LIN {X 0,Y 246.856,Z 370.948,A -85,B 0,C 180,E1 -19029.765,E2 -19029.765} C_VEL
LIN {X 0,Y 247.348,Z 370.564,A -85,B 0,C 180,E1 -19032.995,E2 -19032.995} C_VEL
LIN {X 0,Y 247.895,Z 369.406,A -85,B 0,C 180,E1 -19035.136,E2 -19035.136} C_VEL
LIN {X 0,Y 249.122,Z 366.297,A -85,B 0,C 180,E1 -19038.384,E2 -19038.384} C_VEL
LIN {X 0,Y 250.289,Z 363.157,A -85,B 0,C 180,E1 -19040.597,E2 -19040.597} C_VEL
LIN {X 0,Y 252.077,Z 357.887,A -85,B 0,C 180,E1 -19043.344,E2 -19043.344} C_VEL
LIN {X 0,Y 254.344,Z 351.173,A -85,B 0,C 180,E1 -19045.993,E2 -19045.993} C_VEL
LIN {X 0,Y 256.495,Z 344.263,A -85,B 0,C 180,E1 -19048.149,E2 -19048.149} C_VEL
LIN {X 0,Y 259.318,Z 334.726,A -85,B 0,C 180,E1 -19050.481,E2 -19050.481} C_VEL
LIN {X 0,Y 261.847,Z 325.143,A -85,B 0,C 180,E1 -19052.343,E2 -19052.343} C_VEL
LIN {X 0,Y 264.393,Z 314.469,A -85,B 0,C 180,E1 -19053.979,E2 -19053.979} C_VEL
LIN {X 0,Y 266.72,Z 302.445,A -85,B 0,C 180,E1 -19055.418,E2 -19055.418} C_VEL
LIN {X 0,Y 268.611,Z 289.891,A -85,B 0,C 180,E1 -19056.566,E2 -19056.566} C_VEL
LIN {X 0,Y 269.924,Z 277.78,A -85,B 0,C 180,E1 -19057.366,E2 -19057.366} C_VEL
LIN {X 0,Y 270.894,Z 265.944,A -85,B 0,C 180,E1 -19057.879,E2 -19057.879} C_VEL
LIN {X 0,Y 273.87,Z 206.722,A -85,B 0,C 180,E1 -19059.638,E2 -19059.638} C_VEL
LIN {X 0,Y 268.916,Z 195.841,A -85,B 0,C 180,E1 -19060.94,E2 -19060.94} C_VEL
LIN {X 0,Y 263.621,Z 185.772,A -85,B 0,C 180,E1 -19062.367,E2 -19062.367} C_VEL
LIN {X 0,Y 258.048,Z 176.312,A -85,B 0,C 180,E1 -19063.953,E2 -19063.953} C_VEL
LIN {X 0,Y 254.517,Z 171.077,A -85,B 0,C 180,E1 -19064.995,E2 -19064.995} C_VEL
LIN {X 0,Y 252.04,Z 167.296,A -85,B 0,C 180,E1 -19065.776,E2 -19065.776} C_VEL
LIN {X 0,Y 250.053,Z 164.997,A -85,B 0,C 180,E1 -19066.386,E2 -19066.386} C_VEL
LIN {X 0,Y 249.299,Z 163,A -85,B 0,C 180,E1 -19066.708,E2 -19066.708} C_VEL
LIN {X 0,Y 249.238,Z 162.44,A -85,B 0,C 180,E1 -19067.171,E2 -19067.171} C_VEL
LIN {X 0,Y 249.422,Z 162.416,A -85,B 0,C 180,E1 -19071.902,E2 -19071.902} C_VEL
LIN {X 0,Y 249.267,Z 162.431,A -85,B 0,C 180,E1 -19075.149,E2 -19075.149} C_VEL
LIN {X 0,Y 249.636,Z 162.383,A -85,B 0,C 180,E1 -19078.272,E2 -19078.272} C_VEL
LIN {X 0,Y 249.448,Z 162.41,A -85,B 0,C 180,E1 -19079.172,E2 -19079.172} C_VEL
LIN {X 0,Y 248.655,Z 162.514,A -85,B 0,C 180,E1 -19080.058,E2 -19080.058} C_VEL
LIN {X 0,Y 246.082,Z 162.842,A -85,B 0,C 180,E1 -19081.801,E2 -19081.801} C_VEL
LIN {X 0,Y 243.415,Z 163.173,A -85,B 0,C 180,E1 -19083.583,E2 -19083.583} C_VEL
LIN {X 0,Y 242.311,Z 163.302,A -85,B 0,C 180,E1 -19084.974,E2 -19084.974} C_VEL
LIN {X 0,Y 242.252,Z 163.303,A -85,B 0,C 180,E1 -19085.447,E2 -19085.447} C_VEL
LIN {X 0,Y 242.373,Z 163.288,A -85,B 0,C 180,E1 -19088.337,E2 -19088.337} C_VEL
LIN {X 0,Y 242.112,Z 163.324,A -85,B 0,C 180,E1 -19093.429,E2 -19093.429} C_VEL
LIN {X 0,Y 242.097,Z 163.326,A -85,B 0,C 180,E1 -19096.877,E2 -19096.877} C_VEL
LIN {X 0,Y 241.976,Z 163.342,A -85,B 0,C 180,E1 -19102.184,E2 -19102.184} C_VEL
LIN {X 0,Y 241.991,Z 163.342,A -85,B 0,C 180,E1 -19105.827,E2 -19105.827} C_VEL
LIN {X 0,Y 241.968,Z 163.346,A -85,B 0,C 180,E1 -19109.59,E2 -19109.59} C_VEL
LIN {X 0,Y 241.984,Z 163.343,A -85,B 0,C 180,E1 -19113.493,E2 -19113.493} C_VEL
LIN {X 0,Y 241.992,Z 163.337,A -85,B 0,C 180,E1 -19117.582,E2 -19117.582} C_VEL
LIN {X 0,Y 241.913,Z 163.348,A -85,B 0,C 180,E1 -19121.929,E2 -19121.929} C_VEL
LIN {X 0,Y 241.966,Z 163.485,A -85,B 0,C 180,E1 -19122.861,E2 -19122.861} C_VEL
LIN {X 0,Y 243.695,Z 168.875,A -85,B 0,C 180,E1 -19126.198,E2 -19126.198} C_VEL
LIN {X 0,Y 246.03,Z 176.729,A -85,B 0,C 180,E1 -19130.47,E2 -19130.47} C_VEL
LIN {X 0,Y 248.775,Z 181.528,A -85,B 0,C 180,E1 -19131.44,E2 -19131.44} C_VEL
LIN {X 0,Y 250.887,Z 185.194,A -85,B 0,C 180,E1 -19132.142,E2 -19132.142} C_VEL
LIN {X 0,Y 253.14,Z 189.148,A -85,B 0,C 180,E1 -19132.863,E2 -19132.863} C_VEL
LIN {X 0,Y 258.623,Z 199.785,A -85,B 0,C 180,E1 -19134.545,E2 -19134.545} C_VEL
LIN {X 0,Y 262.961,Z 209.455,A -85,B 0,C 180,E1 -19135.836,E2 -19135.836} C_VEL
LIN {X 0,Y 264.023,Z 212.177,A -85,B 0,C 180,E1 -19136.15,E2 -19136.15} C_VEL
LIN {X 0,Y 266.656,Z 231.739,A -85,B 0,C 180,E1 -19137.415,E2 -19137.415} C_VEL
LIN {X 0,Y 267.038,Z 237.313,A -85,B 0,C 180,E1 -19137.701,E2 -19137.701} C_VEL
LIN {X 0,Y 264.288,Z 288.303,A -85,B 0,C 180,E1 -19139.27,E2 -19139.27} C_VEL
LIN {X 0,Y 262.866,Z 301.195,A -85,B 0,C 180,E1 -19139.913,E2 -19139.913} C_VEL
LIN {X 0,Y 260.719,Z 314.41,A -85,B 0,C 180,E1 -19140.862,E2 -19140.862} C_VEL
LIN {X 0,Y 258.383,Z 326.026,A -85,B 0,C 180,E1 -19142.017,E2 -19142.017} C_VEL
LIN {X 0,Y 256.04,Z 336.044,A -85,B 0,C 180,E1 -19143.289,E2 -19143.289} C_VEL
LIN {X 0,Y 253.243,Z 346.542,A -85,B 0,C 180,E1 -19144.961,E2 -19144.961} C_VEL
LIN {X 0,Y 250.418,Z 356.075,A -85,B 0,C 180,E1 -19146.863,E2 -19146.863} C_VEL
LIN {X 0,Y 247.988,Z 364.065,A -85,B 0,C 180,E1 -19148.86,E2 -19148.86} C_VEL
LIN {X 0,Y 245.836,Z 371.131,A -85,B 0,C 180,E1 -19151.044,E2 -19151.044} C_VEL
LIN {X 0,Y 243.985,Z 376.967,A -85,B 0,C 180,E1 -19153.258,E2 -19153.258} C_VEL
LIN {X 0,Y 242.22,Z 382.172,A -85,B 0,C 180,E1 -19155.721,E2 -19155.721} C_VEL
LIN {X 0,Y 241.046,Z 386.261,A -85,B 0,C 180,E1 -19158.223,E2 -19158.223} C_VEL
LIN {X 0,Y 240.142,Z 390.101,A -85,B 0,C 180,E1 -19161.585,E2 -19161.585} C_VEL
LIN {X 0,Y 239.898,Z 391.414,A -85,B 0,C 180,E1 -19163.269,E2 -19163.269} C_VEL
LIN {X 0,Y 239.808,Z 392.369,A -85,B 0,C 180,E1 -19165.167,E2 -19165.167} C_VEL
LIN {X 0,Y 239.971,Z 392.844,A -85,B 0,C 180,E1 -19168.321,E2 -19168.321} C_VEL
LIN {X 0,Y 240.02,Z 392.522,A -85,B 0,C 180,E1 -19169.999,E2 -19169.999} C_VEL
LIN {X 0,Y 239.988,Z 391.764,A -85,B 0,C 180,E1 -19171.677,E2 -19171.677} C_VEL
LIN {X 0,Y 239.94,Z 390.556,A -85,B 0,C 180,E1 -19173.357,E2 -19173.357} C_VEL
LIN {X 0,Y 239.915,Z 388.833,A -85,B 0,C 180,E1 -19175.126,E2 -19175.126} C_VEL
LIN {X 0,Y 240.072,Z 385.603,A -85,B 0,C 180,E1 -19177.569,E2 -19177.569} C_VEL
LIN {X 0,Y 240.467,Z 381.156,A -85,B 0,C 180,E1 -19180.099,E2 -19180.099} C_VEL
LIN {X 0,Y 241.155,Z 375.461,A -85,B 0,C 180,E1 -19182.624,E2 -19182.624} C_VEL
LIN {X 0,Y 242.422,Z 368.321,A -85,B 0,C 180,E1 -19185.124,E2 -19185.124} C_VEL
LIN {X 0,Y 243.817,Z 359.891,A -85,B 0,C 180,E1 -19187.472,E2 -19187.472} C_VEL
LIN {X 0,Y 245.472,Z 350.125,A -85,B 0,C 180,E1 -19189.657,E2 -19189.657} C_VEL
LIN {X 0,Y 247.269,Z 339.949,A -85,B 0,C 180,E1 -19191.464,E2 -19191.464} C_VEL
LIN {X 0,Y 249.026,Z 328.652,A -85,B 0,C 180,E1 -19193.052,E2 -19193.052} C_VEL
LIN {X 0,Y 250.727,Z 316.016,A -85,B 0,C 180,E1 -19194.421,E2 -19194.421} C_VEL
LIN {X 0,Y 252.123,Z 303.843,A -85,B 0,C 180,E1 -19195.377,E2 -19195.377} C_VEL
LIN {X 0,Y 253.166,Z 290.677,A -85,B 0,C 180,E1 -19196.092,E2 -19196.092} C_VEL
LIN {X 0,Y 254.777,Z 250.055,A -85,B 0,C 180,E1 -19197.365,E2 -19197.365} C_VEL
LIN {X 0,Y 255.305,Z 232.614,A -85,B 0,C 180,E1 -19197.902,E2 -19197.902} C_VEL
LIN {X 0,Y 250.199,Z 193.129,A -85,B 0,C 180,E1 -19199.733,E2 -19199.733} C_VEL
LIN {X 0,Y 245.773,Z 180.605,A -85,B 0,C 180,E1 -19200.64,E2 -19200.64} C_VEL
LIN {X 0,Y 243.127,Z 168.039,A -85,B 0,C 180,E1 -19205.318,E2 -19205.318} C_VEL
LIN {X 0,Y 242.041,Z 163.337,A -85,B 0,C 180,E1 -19207.221,E2 -19207.221} C_VEL
LIN {X 0,Y 241.938,Z 163.352,A -85,B 0,C 180,E1 -19211.921,E2 -19211.921} C_VEL
LIN {X 0,Y 241.934,Z 163.348,A -85,B 0,C 180,E1 -19216.57,E2 -19216.57} C_VEL
LIN {X 0,Y 241.956,Z 163.345,A -85,B 0,C 180,E1 -19220.28,E2 -19220.28} C_VEL
LIN {X 0,Y 242.004,Z 163.339,A -85,B 0,C 180,E1 -19224.491,E2 -19224.491} C_VEL
LIN {X 0,Y 241.975,Z 163.343,A -85,B 0,C 180,E1 -19228.479,E2 -19228.479} C_VEL
LIN {X 0,Y 242.009,Z 163.337,A -85,B 0,C 180,E1 -19232.312,E2 -19232.312} C_VEL
LIN {X 0,Y 242.056,Z 163.327,A -85,B 0,C 180,E1 -19236.015,E2 -19236.015} C_VEL
LIN {X 0,Y 242.025,Z 163.338,A -85,B 0,C 180,E1 -19239.606,E2 -19239.606} C_VEL
LIN {X 0,Y 242.114,Z 163.321,A -85,B 0,C 180,E1 -19243.315,E2 -19243.315} C_VEL
LIN {X 0,Y 242.182,Z 163.316,A -85,B 0,C 180,E1 -19248.279,E2 -19248.279} C_VEL
LIN {X 0,Y 242.424,Z 163.278,A -85,B 0,C 180,E1 -19251.665,E2 -19251.665} C_VEL
LIN {X 0,Y 242.258,Z 163.307,A -85,B 0,C 180,E1 -19255.006,E2 -19255.006} C_VEL
LIN {X 0,Y 242.635,Z 163.26,A -85,B 0,C 180,E1 -19258.339,E2 -19258.339} C_VEL
LIN {X 0,Y 242.634,Z 163.251,A -85,B 0,C 180,E1 -19261.659,E2 -19261.659} C_VEL
LIN {X 0,Y 242.426,Z 163.287,A -85,B 0,C 180,E1 -19266.703,E2 -19266.703} C_VEL
LIN {X 0,Y 242.311,Z 163.299,A -85,B 0,C 180,E1 -19270.021,E2 -19270.021} C_VEL
LIN {X 0,Y 242.163,Z 163.312,A -85,B 0,C 180,E1 -19275.14,E2 -19275.14} C_VEL
LIN {X 0,Y 242.07,Z 163.332,A -85,B 0,C 180,E1 -19278.623,E2 -19278.623} C_VEL
LIN {X 0,Y 242.038,Z 163.334,A -85,B 0,C 180,E1 -19282.176,E2 -19282.176} C_VEL
LIN {X 0,Y 242.062,Z 163.318,A -85,B 0,C 180,E1 -19285.838,E2 -19285.838} C_VEL
LIN {X 0,Y 242.026,Z 163.332,A -85,B 0,C 180,E1 -19289.58,E2 -19289.58} C_VEL
LIN {X 0,Y 241.987,Z 163.336,A -85,B 0,C 180,E1 -19293.49,E2 -19293.49} C_VEL
LIN {X 0,Y 242.015,Z 163.328,A -85,B 0,C 180,E1 -19297.576,E2 -19297.576} C_VEL
LIN {X 0,Y 242.038,Z 163.335,A -85,B 0,C 180,E1 -19301.9,E2 -19301.9} C_VEL
LIN {X 0,Y 242.02,Z 163.33,A -85,B 0,C 180,E1 -19306.548,E2 -19306.548} C_VEL
LIN {X 0,Y 242.024,Z 163.336,A -85,B 0,C 180,E1 -19310.295,E2 -19310.295} C_VEL
LIN {X 0,Y 242.032,Z 163.328,A -85,B 0,C 180,E1 -19314.498,E2 -19314.498} C_VEL
LIN {X 0,Y 241.971,Z 163.342,A -85,B 0,C 180,E1 -19318.48,E2 -19318.48} C_VEL
LIN {X 0,Y 242.004,Z 163.338,A -85,B 0,C 180,E1 -19322.313,E2 -19322.313} C_VEL
LIN {X 0,Y 242.053,Z 163.333,A -85,B 0,C 180,E1 -19326.016,E2 -19326.016} C_VEL
LIN {X 0,Y 242.033,Z 163.337,A -85,B 0,C 180,E1 -19329.609,E2 -19329.609} C_VEL
LIN {X 0,Y 242.159,Z 163.323,A -85,B 0,C 180,E1 -19333.279,E2 -19333.279} C_VEL
LIN {X 0,Y 242.183,Z 163.318,A -85,B 0,C 180,E1 -19338.281,E2 -19338.281} C_VEL
LIN {X 0,Y 242.431,Z 163.288,A -85,B 0,C 180,E1 -19341.667,E2 -19341.667} C_VEL
LIN {X 0,Y 242.259,Z 163.311,A -85,B 0,C 180,E1 -19345.008,E2 -19345.008} C_VEL
LIN {X 0,Y 242.634,Z 163.261,A -85,B 0,C 180,E1 -19348.341,E2 -19348.341} C_VEL
LIN {X 0,Y 242.634,Z 163.261,A -85,B 0,C 180,E1 -19351.661,E2 -19351.661} C_VEL
LIN {X 0,Y 242.416,Z 163.29,A -85,B 0,C 180,E1 -19357.183,E2 -19357.183} C_VEL
LIN {X 0,Y 243.5,Z 166.231,A -85,B 0,C 180,E1 -19357.438,E2 -19357.438} C_VEL
LIN {X 0,Y 250.973,Z 183.621,A -85,B 0,C 180,E1 -19358.835,E2 -19358.835} C_VEL
LIN {X 0,Y 256.265,Z 198.404,A -85,B 0,C 180,E1 -19359.848,E2 -19359.848} C_VEL
LIN {X 0,Y 253.616,Z 268.159,A -85,B 0,C 180,E1 -19361.996,E2 -19361.996} C_VEL
LIN {X 0,Y 252.675,Z 281.492,A -85,B 0,C 180,E1 -19362.723,E2 -19362.723} C_VEL
LIN {X 0,Y 251.611,Z 294.331,A -85,B 0,C 180,E1 -19363.766,E2 -19363.766} C_VEL
LIN {X 0,Y 250.2,Z 306.198,A -85,B 0,C 180,E1 -19365.061,E2 -19365.061} C_VEL
LIN {X 0,Y 248.544,Z 317.502,A -85,B 0,C 180,E1 -19366.638,E2 -19366.638} C_VEL
LIN {X 0,Y 246.824,Z 327.773,A -85,B 0,C 180,E1 -19368.442,E2 -19368.442} C_VEL
LIN {X 0,Y 245.209,Z 337.341,A -85,B 0,C 180,E1 -19370.556,E2 -19370.556} C_VEL
LIN {X 0,Y 243.795,Z 345.266,A -85,B 0,C 180,E1 -19372.711,E2 -19372.711} C_VEL
LIN {X 0,Y 242.442,Z 352.962,A -85,B 0,C 180,E1 -19375.315,E2 -19375.315} C_VEL
LIN {X 0,Y 241.421,Z 358.656,A -85,B 0,C 180,E1 -19377.761,E2 -19377.761} C_VEL
LIN {X 0,Y 240.608,Z 363.958,A -85,B 0,C 180,E1 -19380.742,E2 -19380.742} C_VEL
LIN {X 0,Y 239.939,Z 367.864,A -85,B 0,C 180,E1 -19383.817,E2 -19383.817} C_VEL
LIN {X 0,Y 239.728,Z 369.62,A -85,B 0,C 180,E1 -19385.898,E2 -19385.898} C_VEL
LIN {X 0,Y 239.652,Z 370.797,A -85,B 0,C 180,E1 -19388.014,E2 -19388.014} C_VEL
LIN {X 0,Y 239.809,Z 371.334,A -85,B 0,C 180,E1 -19390.363,E2 -19390.363} C_VEL
LIN {X 0,Y 240.26,Z 370.996,A -85,B 0,C 180,E1 -19393.007,E2 -19393.007} C_VEL
LIN {X 0,Y 240.933,Z 369.713,A -85,B 0,C 180,E1 -19395.568,E2 -19395.568} C_VEL
LIN {X 0,Y 242.293,Z 366.515,A -85,B 0,C 180,E1 -19398.954,E2 -19398.954} C_VEL
LIN {X 0,Y 244.033,Z 361.975,A -85,B 0,C 180,E1 -19402.042,E2 -19402.042} C_VEL
LIN {X 0,Y 246.091,Z 356.398,A -85,B 0,C 180,E1 -19404.785,E2 -19404.785} C_VEL
LIN {X 0,Y 248.697,Z 349.008,A -85,B 0,C 180,E1 -19407.527,E2 -19407.527} C_VEL
LIN {X 0,Y 251.218,Z 341.32,A -85,B 0,C 180,E1 -19409.765,E2 -19409.765} C_VEL
LIN {X 0,Y 253.797,Z 332.678,A -85,B 0,C 180,E1 -19411.78,E2 -19411.78} C_VEL
LIN {X 0,Y 256.518,Z 322.579,A -85,B 0,C 180,E1 -19413.646,E2 -19413.646} C_VEL
LIN {X 0,Y 259.316,Z 310.658,A -85,B 0,C 180,E1 -19415.375,E2 -19415.375} C_VEL
LIN {X 0,Y 261.448,Z 299.381,A -85,B 0,C 180,E1 -19416.642,E2 -19416.642} C_VEL
LIN {X 0,Y 263.307,Z 286.431,A -85,B 0,C 180,E1 -19417.749,E2 -19417.749} C_VEL
LIN {X 0,Y 264.683,Z 273.244,A -85,B 0,C 180,E1 -19418.529,E2 -19418.529} C_VEL
LIN {X 0,Y 265.814,Z 256.165,A -85,B 0,C 180,E1 -19419.114,E2 -19419.114} C_VEL
LIN {X 0,Y 268.28,Z 208.894,A -85,B 0,C 180,E1 -19420.539,E2 -19420.539} C_VEL
LIN {X 0,Y 263.182,Z 197.855,A -85,B 0,C 180,E1 -19421.947,E2 -19421.947} C_VEL
LIN {X 0,Y 256.603,Z 185.498,A -85,B 0,C 180,E1 -19423.86,E2 -19423.86} C_VEL
LIN {X 0,Y 250.777,Z 176.379,A -85,B 0,C 180,E1 -19425.651,E2 -19425.651} C_VEL
LIN {X 0,Y 248.175,Z 172.649,A -85,B 0,C 180,E1 -19426.49,E2 -19426.49} C_VEL
LIN {X 0,Y 245.905,Z 169.455,A -85,B 0,C 180,E1 -19427.246,E2 -19427.246} C_VEL
LIN {X 0,Y 245.166,Z 168.24,A -85,B 0,C 180,E1 -19427.513,E2 -19427.513} C_VEL
LIN {X 0,Y 243.09,Z 165.951,A -85,B 0,C 180,E1 -19428.22,E2 -19428.22} C_VEL
LIN {X 0,Y 242.265,Z 163.59,A -85,B 0,C 180,E1 -19428.603,E2 -19428.603} C_VEL
LIN {X 0,Y 242.221,Z 163.314,A -85,B 0,C 180,E1 -19429.13,E2 -19429.13} C_VEL
LIN {X 0,Y 242.376,Z 163.295,A -85,B 0,C 180,E1 -19431.665,E2 -19431.665} C_VEL
LIN {X 0,Y 242.401,Z 163.291,A -85,B 0,C 180,E1 -19433.341,E2 -19433.341} C_VEL
LIN {X 0,Y 242.622,Z 163.257,A -85,B 0,C 180,E1 -19438.341,E2 -19438.341} C_VEL
LIN {X 0,Y 242.619,Z 163.26,A -85,B 0,C 180,E1 -19441.661,E2 -19441.661} C_VEL
LIN {X 0,Y 242.252,Z 163.303,A -85,B 0,C 180,E1 -19445.447,E2 -19445.447} C_VEL
LIN {X 0,Y 241.65,Z 163.373,A -85,B 0,C 180,E1 -19446.836,E2 -19446.836} C_VEL
LIN {X 0,Y 240.066,Z 163.577,A -85,B 0,C 180,E1 -19448.199,E2 -19448.199} C_VEL
LIN {X 0,Y 236.239,Z 164.051,A -85,B 0,C 180,E1 -19450.942,E2 -19450.942} C_VEL
LIN {X 0,Y 235.141,Z 164.187,A -85,B 0,C 180,E1 -19452.376,E2 -19452.376} C_VEL
LIN {X 0,Y 235.045,Z 164.194,A -85,B 0,C 180,E1 -19452.862,E2 -19452.862} C_VEL
LIN {X 0,Y 235.055,Z 164.203,A -85,B 0,C 180,E1 -19456.903,E2 -19456.903} C_VEL
LIN {X 0,Y 234.961,Z 164.217,A -85,B 0,C 180,E1 -19461.987,E2 -19461.987} C_VEL
LIN {X 0,Y 234.927,Z 164.215,A -85,B 0,C 180,E1 -19466.664,E2 -19466.664} C_VEL
LIN {X 0,Y 234.9,Z 164.218,A -85,B 0,C 180,E1 -19470.573,E2 -19470.573} C_VEL
LIN {X 0,Y 234.934,Z 164.212,A -85,B 0,C 180,E1 -19474.638,E2 -19474.638} C_VEL
LIN {X 0,Y 234.917,Z 164.217,A -85,B 0,C 180,E1 -19478.935,E2 -19478.935} C_VEL
LIN {X 0,Y 234.904,Z 164.425,A -85,B 0,C 180,E1 -19480.88,E2 -19480.88} C_VEL
LIN {X 0,Y 237.096,Z 171.042,A -85,B 0,C 180,E1 -19485.351,E2 -19485.351} C_VEL
LIN {X 0,Y 238.745,Z 176.397,A -85,B 0,C 180,E1 -19488.409,E2 -19488.409} C_VEL
LIN {X 0,Y 241.757,Z 181.355,A -85,B 0,C 180,E1 -19489.56,E2 -19489.56} C_VEL
LIN {X 0,Y 243.391,Z 184.153,A -85,B 0,C 180,E1 -19490.167,E2 -19490.167} C_VEL
LIN {X 0,Y 246.439,Z 189.214,A -85,B 0,C 180,E1 -19491.224,E2 -19491.224} C_VEL
LIN {X 0,Y 250.836,Z 197.293,A -85,B 0,C 180,E1 -19492.705,E2 -19492.705} C_VEL
LIN {X 0,Y 256.982,Z 210.263,A -85,B 0,C 180,E1 -19494.654,E2 -19494.654} C_VEL
LIN {X 0,Y 259.057,Z 215.917,A -85,B 0,C 180,E1 -19495.329,E2 -19495.329} C_VEL
LIN {X 0,Y 261.248,Z 233.871,A -85,B 0,C 180,E1 -19496.508,E2 -19496.508} C_VEL
LIN {X 0,Y 261.539,Z 238.959,A -85,B 0,C 180,E1 -19496.77,E2 -19496.77} C_VEL
LIN {X 0,Y 258.697,Z 288.182,A -85,B 0,C 180,E1 -19498.306,E2 -19498.306} C_VEL
LIN {X 0,Y 257.222,Z 300.955,A -85,B 0,C 180,E1 -19498.954,E2 -19498.954} C_VEL
LIN {X 0,Y 255.004,Z 314.123,A -85,B 0,C 180,E1 -19499.916,E2 -19499.916} C_VEL
LIN {X 0,Y 252.191,Z 327.24,A -85,B 0,C 180,E1 -19501.266,E2 -19501.266} C_VEL
LIN {X 0,Y 249.779,Z 336.941,A -85,B 0,C 180,E1 -19502.564,E2 -19502.564} C_VEL
LIN {X 0,Y 246.856,Z 347.196,A -85,B 0,C 180,E1 -19504.267,E2 -19504.267} C_VEL
LIN {X 0,Y 243.914,Z 356.501,A -85,B 0,C 180,E1 -19506.209,E2 -19506.209} C_VEL
LIN {X 0,Y 240.995,Z 365.586,A -85,B 0,C 180,E1 -19508.62,E2 -19508.62} C_VEL
LIN {X 0,Y 238.534,Z 372.957,A -85,B 0,C 180,E1 -19511.088,E2 -19511.088} C_VEL
LIN {X 0,Y 236.524,Z 378.907,A -85,B 0,C 180,E1 -19513.603,E2 -19513.603} C_VEL
LIN {X 0,Y 234.799,Z 383.635,A -85,B 0,C 180,E1 -19516.145,E2 -19516.145} C_VEL
LIN {X 0,Y 233.762,Z 387.273,A -85,B 0,C 180,E1 -19518.73,E2 -19518.73} C_VEL
LIN {X 0,Y 233.09,Z 389.922,A -85,B 0,C 180,E1 -19521.328,E2 -19521.328} C_VEL
LIN {X 0,Y 232.819,Z 391.19,A -85,B 0,C 180,E1 -19523.064,E2 -19523.064} C_VEL
LIN {X 0,Y 232.719,Z 392.172,A -85,B 0,C 180,E1 -19525.272,E2 -19525.272} C_VEL
LIN {X 0,Y 232.897,Z 392.499,A -85,B 0,C 180,E1 -19528.27,E2 -19528.27} C_VEL
LIN {X 0,Y 232.948,Z 392.138,A -85,B 0,C 180,E1 -19529.999,E2 -19529.999} C_VEL
LIN {X 0,Y 232.917,Z 391.316,A -85,B 0,C 180,E1 -19531.728,E2 -19531.728} C_VEL
LIN {X 0,Y 232.858,Z 390.072,A -85,B 0,C 180,E1 -19533.46,E2 -19533.46} C_VEL
LIN {X 0,Y 232.841,Z 387.374,A -85,B 0,C 180,E1 -19536.063,E2 -19536.063} C_VEL
LIN {X 0,Y 233.143,Z 383.613,A -85,B 0,C 180,E1 -19538.668,E2 -19538.668} C_VEL
LIN {X 0,Y 233.641,Z 378.67,A -85,B 0,C 180,E1 -19541.274,E2 -19541.274} C_VEL
LIN {X 0,Y 234.605,Z 372.417,A -85,B 0,C 180,E1 -19543.865,E2 -19543.865} C_VEL
LIN {X 0,Y 235.978,Z 364.596,A -85,B 0,C 180,E1 -19546.434,E2 -19546.434} C_VEL
LIN {X 0,Y 237.534,Z 355.633,A -85,B 0,C 180,E1 -19548.772,E2 -19548.772} C_VEL
LIN {X 0,Y 239.34,Z 345.658,A -85,B 0,C 180,E1 -19550.856,E2 -19550.856} C_VEL
LIN {X 0,Y 241.052,Z 335.864,A -85,B 0,C 180,E1 -19552.498,E2 -19552.498} C_VEL
LIN {X 0,Y 242.723,Z 325.281,A -85,B 0,C 180,E1 -19553.913,E2 -19553.913} C_VEL
LIN {X 0,Y 244.427,Z 312.638,A -85,B 0,C 180,E1 -19555.207,E2 -19555.207} C_VEL
LIN {X 0,Y 245.806,Z 299.367,A -85,B 0,C 180,E1 -19556.191,E2 -19556.191} C_VEL
LIN {X 0,Y 246.761,Z 285.995,A -85,B 0,C 180,E1 -19556.823,E2 -19556.823} C_VEL
LIN {X 0,Y 248.696,Z 233.355,A -85,B 0,C 180,E1 -19558.477,E2 -19558.477} C_VEL
LIN {X 0,Y 243.803,Z 195.193,A -85,B 0,C 180,E1 -19560.307,E2 -19560.307} C_VEL
LIN {X 0,Y 238.46,Z 180.289,A -85,B 0,C 180,E1 -19561.437,E2 -19561.437} C_VEL
LIN {X 0,Y 236.274,Z 169.835,A -85,B 0,C 180,E1 -19565.451,E2 -19565.451} C_VEL
LIN {X 0,Y 234.974,Z 164.217,A -85,B 0,C 180,E1 -19567.707,E2 -19567.707} C_VEL
LIN {X 0,Y 234.884,Z 164.231,A -85,B 0,C 180,E1 -19571.579,E2 -19571.579} C_VEL
LIN {X 0,Y 234.895,Z 164.226,A -85,B 0,C 180,E1 -19575.894,E2 -19575.894} C_VEL
LIN {X 0,Y 234.883,Z 164.225,A -85,B 0,C 180,E1 -19578.831,E2 -19578.831} C_VEL
LIN {X 0,Y 234.918,Z 164.222,A -85,B 0,C 180,E1 -19581.077,E2 -19581.077} C_VEL
LIN {X 0,Y 234.941,Z 164.22,A -85,B 0,C 180,E1 -19585.363,E2 -19585.363} C_VEL
LIN {X 0,Y 234.931,Z 164.22,A -85,B 0,C 180,E1 -19589.431,E2 -19589.431} C_VEL
LIN {X 0,Y 234.993,Z 164.212,A -85,B 0,C 180,E1 -19593.792,E2 -19593.792} C_VEL
LIN {X 0,Y 235.005,Z 164.211,A -85,B 0,C 180,E1 -19598.968,E2 -19598.968} C_VEL
LIN {X 0,Y 235.077,Z 164.196,A -85,B 0,C 180,E1 -19604.39,E2 -19604.39} C_VEL
LIN {X 0,Y 235.236,Z 164.179,A -85,B 0,C 180,E1 -19609.672,E2 -19609.672} C_VEL
LIN {X 0,Y 235.401,Z 164.156,A -85,B 0,C 180,E1 -19613.14,E2 -19613.14} C_VEL
LIN {X 0,Y 235.594,Z 164.137,A -85,B 0,C 180,E1 -19618.29,E2 -19618.29} C_VEL
LIN {X 0,Y 235.594,Z 164.127,A -85,B 0,C 180,E1 -19621.708,E2 -19621.708} C_VEL
LIN {X 0,Y 235.4,Z 164.164,A -85,B 0,C 180,E1 -19626.858,E2 -19626.858} C_VEL
LIN {X 0,Y 235.235,Z 164.182,A -85,B 0,C 180,E1 -19630.326,E2 -19630.326} C_VEL
LIN {X 0,Y 235.11,Z 164.19,A -85,B 0,C 180,E1 -19635.606,E2 -19635.606} C_VEL
LIN {X 0,Y 235.005,Z 164.209,A -85,B 0,C 180,E1 -19639.205,E2 -19639.205} C_VEL
LIN {X 0,Y 234.973,Z 164.209,A -85,B 0,C 180,E1 -19642.881,E2 -19642.881} C_VEL
LIN {X 0,Y 234.966,Z 164.207,A -85,B 0,C 180,E1 -19646.657,E2 -19646.657} C_VEL
LIN {X 0,Y 234.928,Z 164.219,A -85,B 0,C 180,E1 -19650.567,E2 -19650.567} C_VEL
LIN {X 0,Y 234.956,Z 164.208,A -85,B 0,C 180,E1 -19654.632,E2 -19654.632} C_VEL
LIN {X 0,Y 234.992,Z 164.207,A -85,B 0,C 180,E1 -19658.961,E2 -19658.961} C_VEL
LIN {X 0,Y 234.992,Z 164.21,A -85,B 0,C 180,E1 -19663.46,E2 -19663.46} C_VEL
LIN {X 0,Y 234.998,Z 164.21,A -85,B 0,C 180,E1 -19668.387,E2 -19668.387} C_VEL
LIN {X 0,Y 234.981,Z 164.213,A -85,B 0,C 180,E1 -19671.092,E2 -19671.092} C_VEL
LIN {X 0,Y 234.956,Z 164.211,A -85,B 0,C 180,E1 -19675.367,E2 -19675.367} C_VEL
LIN {X 0,Y 234.964,Z 164.215,A -85,B 0,C 180,E1 -19680.158,E2 -19680.158} C_VEL
LIN {X 0,Y 234.989,Z 164.214,A -85,B 0,C 180,E1 -19683.794,E2 -19683.794} C_VEL
LIN {X 0,Y 235.007,Z 164.212,A -85,B 0,C 180,E1 -19688.97,E2 -19688.97} C_VEL
LIN {X 0,Y 235.092,Z 164.202,A -85,B 0,C 180,E1 -19693.06,E2 -19693.06} C_VEL
LIN {X 0,Y 235.143,Z 164.196,A -85,B 0,C 180,E1 -19697.925,E2 -19697.925} C_VEL
LIN {X 0,Y 235.387,Z 164.167,A -85,B 0,C 180,E1 -19701.415,E2 -19701.415} C_VEL
LIN {X 0,Y 235.402,Z 164.167,A -85,B 0,C 180,E1 -19703.142,E2 -19703.142} C_VEL
LIN {X 0,Y 235.593,Z 164.138,A -85,B 0,C 180,E1 -19708.292,E2 -19708.292} C_VEL
LIN {X 0,Y 235.593,Z 164.138,A -85,B 0,C 180,E1 -19711.71,E2 -19711.71} C_VEL
LIN {X 0,Y 235.359,Z 164.169,A -85,B 0,C 180,E1 -19716.43,E2 -19716.43} C_VEL
LIN {X 0,Y 236.439,Z 167.089,A -85,B 0,C 180,E1 -19716.675,E2 -19716.675} C_VEL
LIN {X 0,Y 243.5,Z 182.958,A -85,B 0,C 180,E1 -19718.04,E2 -19718.04} C_VEL
LIN {X 0,Y 249.65,Z 199.841,A -85,B 0,C 180,E1 -19719.265,E2 -19719.265} C_VEL
LIN {X 0,Y 246.975,Z 268.023,A -85,B 0,C 180,E1 -19721.415,E2 -19721.415} C_VEL
LIN {X 0,Y 245.998,Z 281.897,A -85,B 0,C 180,E1 -19722.19,E2 -19722.19} C_VEL
LIN {X 0,Y 244.851,Z 294.888,A -85,B 0,C 180,E1 -19723.276,E2 -19723.276} C_VEL
LIN {X 0,Y 243.365,Z 306.967,A -85,B 0,C 180,E1 -19724.638,E2 -19724.638} C_VEL
LIN {X 0,Y 241.617,Z 318.399,A -85,B 0,C 180,E1 -19726.288,E2 -19726.288} C_VEL
LIN {X 0,Y 239.875,Z 328.509,A -85,B 0,C 180,E1 -19728.138,E2 -19728.138} C_VEL
LIN {X 0,Y 238.107,Z 338.524,A -85,B 0,C 180,E1 -19730.44,E2 -19730.44} C_VEL
LIN {X 0,Y 236.55,Z 347.149,A -85,B 0,C 180,E1 -19732.927,E2 -19732.927} C_VEL
LIN {X 0,Y 235.238,Z 354.064,A -85,B 0,C 180,E1 -19735.437,E2 -19735.437} C_VEL
LIN {X 0,Y 234.329,Z 359.113,A -85,B 0,C 180,E1 -19737.703,E2 -19737.703} C_VEL
LIN {X 0,Y 233.491,Z 364.396,A -85,B 0,C 180,E1 -19740.778,E2 -19740.778} C_VEL
LIN {X 0,Y 232.829,Z 368.27,A -85,B 0,C 180,E1 -19743.948,E2 -19743.948} C_VEL
LIN {X 0,Y 232.556,Z 370.658,A -85,B 0,C 180,E1 -19747.188,E2 -19747.188} C_VEL
LIN {X 0,Y 232.635,Z 371.499,A -85,B 0,C 180,E1 -19749.378,E2 -19749.378} C_VEL
LIN {X 0,Y 232.864,Z 371.647,A -85,B 0,C 180,E1 -19751.605,E2 -19751.605} C_VEL
LIN {X 0,Y 233.374,Z 371.16,A -85,B 0,C 180,E1 -19753.841,E2 -19753.841} C_VEL
LIN {X 0,Y 234.076,Z 369.838,A -85,B 0,C 180,E1 -19756.327,E2 -19756.327} C_VEL
LIN {X 0,Y 235.596,Z 366.555,A -85,B 0,C 180,E1 -19759.726,E2 -19759.726} C_VEL
LIN {X 0,Y 236.968,Z 363.161,A -85,B 0,C 180,E1 -19762.138,E2 -19762.138} C_VEL
LIN {X 0,Y 238.714,Z 358.835,A -85,B 0,C 180,E1 -19764.491,E2 -19764.491} C_VEL
LIN {X 0,Y 240.785,Z 353.417,A -85,B 0,C 180,E1 -19766.817,E2 -19766.817} C_VEL
LIN {X 0,Y 243.568,Z 345.609,A -85,B 0,C 180,E1 -19769.45,E2 -19769.45} C_VEL
LIN {X 0,Y 246.375,Z 337.278,A -85,B 0,C 180,E1 -19771.659,E2 -19771.659} C_VEL
LIN {X 0,Y 248.995,Z 328.529,A -85,B 0,C 180,E1 -19773.522,E2 -19773.522} C_VEL
LIN {X 0,Y 251.895,Z 317.824,A -85,B 0,C 180,E1 -19775.328,E2 -19775.328} C_VEL
LIN {X 0,Y 254.535,Z 305.951,A -85,B 0,C 180,E1 -19776.908,E2 -19776.908} C_VEL
LIN {X 0,Y 256.752,Z 293.52,A -85,B 0,C 180,E1 -19778.15,E2 -19778.15} C_VEL
LIN {X 0,Y 258.399,Z 281.161,A -85,B 0,C 180,E1 -19779.066,E2 -19779.066} C_VEL
LIN {X 0,Y 259.503,Z 269.649,A -85,B 0,C 180,E1 -19779.651,E2 -19779.651} C_VEL
LIN {X 0,Y 262.857,Z 211.398,A -85,B 0,C 180,E1 -19781.445,E2 -19781.445} C_VEL
LIN {X 0,Y 257.263,Z 199.274,A -85,B 0,C 180,E1 -19783.109,E2 -19783.109} C_VEL
LIN {X 0,Y 251.148,Z 188.18,A -85,B 0,C 180,E1 -19784.994,E2 -19784.994} C_VEL
LIN {X 0,Y 246.432,Z 180.763,A -85,B 0,C 180,E1 -19786.537,E2 -19786.537} C_VEL
LIN {X 0,Y 244.385,Z 177.876,A -85,B 0,C 180,E1 -19787.225,E2 -19787.225} C_VEL
LIN {X 0,Y 241.531,Z 173.769,A -85,B 0,C 180,E1 -19788.249,E2 -19788.249} C_VEL
LIN {X 0,Y 239.352,Z 170.876,A -85,B 0,C 180,E1 -19789.052,E2 -19789.052} C_VEL
LIN {X 0,Y 238.526,Z 169.349,A -85,B 0,C 180,E1 -19789.389,E2 -19789.389} C_VEL
LIN {X 0,Y 236.453,Z 167.322,A -85,B 0,C 180,E1 -19790.164,E2 -19790.164} C_VEL
LIN {X 0,Y 235.374,Z 164.585,A -85,B 0,C 180,E1 -19790.682,E2 -19790.682} C_VEL
LIN {X 0,Y 235.307,Z 164.18,A -85,B 0,C 180,E1 -19790.799,E2 -19790.799} C_VEL
LIN {X 0,Y 235.352,Z 164.167,A -85,B 0,C 180,E1 -19793.141,E2 -19793.141} C_VEL
LIN {X 0,Y 235.581,Z 164.135,A -85,B 0,C 180,E1 -19798.291,E2 -19798.291} C_VEL
LIN {X 0,Y 235.578,Z 164.136,A -85,B 0,C 180,E1 -19801.71,E2 -19801.71} C_VEL
LIN {X 0,Y 235.352,Z 164.155,A -85,B 0,C 180,E1 -19806.861,E2 -19806.861} C_VEL
LIN {X 0,Y 235.188,Z 164.176,A -85,B 0,C 180,E1 -19810.33,E2 -19810.33} C_VEL
LIN {X 0,Y 235.045,Z 164.194,A -85,B 0,C 180,E1 -19812.862,E2 -19812.862} C_VEL
LIN {X 0,Y 234.349,Z 164.286,A -85,B 0,C 180,E1 -19814.293,E2 -19814.293} C_VEL
LIN {X 0,Y 231.449,Z 164.648,A -85,B 0,C 180,E1 -19816.625,E2 -19816.625} C_VEL
LIN {X 0,Y 228.999,Z 164.95,A -85,B 0,C 180,E1 -19818.527,E2 -19818.527} C_VEL
LIN {X 0,Y 227.954,Z 165.077,A -85,B 0,C 180,E1 -19820.005,E2 -19820.005} C_VEL
LIN {X 0,Y 227.872,Z 165.089,A -85,B 0,C 180,E1 -19820.506,E2 -19820.506} C_VEL
LIN {X 0,Y 227.86,Z 165.089,A -85,B 0,C 180,E1 -19823.64,E2 -19823.64} C_VEL
LIN {X 0,Y 227.846,Z 165.092,A -85,B 0,C 180,E1 -19827.561,E2 -19827.561} C_VEL
LIN {X 0,Y 227.859,Z 165.091,A -85,B 0,C 180,E1 -19831.625,E2 -19831.625} C_VEL
LIN {X 0,Y 227.886,Z 165.092,A -85,B 0,C 180,E1 -19835.872,E2 -19835.872} C_VEL
LIN {X 0,Y 227.884,Z 165.232,A -85,B 0,C 180,E1 -19838.496,E2 -19838.496} C_VEL
LIN {X 0,Y 230.002,Z 171.808,A -85,B 0,C 180,E1 -19843.434,E2 -19843.434} C_VEL
LIN {X 0,Y 231.328,Z 175.779,A -85,B 0,C 180,E1 -19845.954,E2 -19845.954} C_VEL
LIN {X 0,Y 234.254,Z 180.515,A -85,B 0,C 180,E1 -19847.232,E2 -19847.232} C_VEL
LIN {X 0,Y 235.608,Z 182.469,A -85,B 0,C 180,E1 -19847.784,E2 -19847.784} C_VEL
LIN {X 0,Y 239.771,Z 189.402,A -85,B 0,C 180,E1 -19849.424,E2 -19849.424} C_VEL
LIN {X 0,Y 242.83,Z 194.654,A -85,B 0,C 180,E1 -19850.553,E2 -19850.553} C_VEL
LIN {X 0,Y 247.503,Z 203.716,A -85,B 0,C 180,E1 -19852.203,E2 -19852.203} C_VEL
LIN {X 0,Y 252.588,Z 214.778,A -85,B 0,C 180,E1 -19853.906,E2 -19853.906} C_VEL
LIN {X 0,Y 254.013,Z 218.79,A -85,B 0,C 180,E1 -19854.395,E2 -19854.395} C_VEL
LIN {X 0,Y 255.959,Z 235.764,A -85,B 0,C 180,E1 -19855.547,E2 -19855.547} C_VEL
LIN {X 0,Y 256.137,Z 240.08,A -85,B 0,C 180,E1 -19855.77,E2 -19855.77} C_VEL
LIN {X 0,Y 253.197,Z 287.954,A -85,B 0,C 180,E1 -19857.296,E2 -19857.296} C_VEL
LIN {X 0,Y 251.568,Z 301.427,A -85,B 0,C 180,E1 -19857.998,E2 -19857.998} C_VEL
LIN {X 0,Y 249.525,Z 312.819,A -85,B 0,C 180,E1 -19858.831,E2 -19858.831} C_VEL
LIN {X 0,Y 246.825,Z 325.388,A -85,B 0,C 180,E1 -19860.112,E2 -19860.112} C_VEL
LIN {X 0,Y 243.835,Z 336.653,A -85,B 0,C 180,E1 -19861.602,E2 -19861.602} C_VEL
LIN {X 0,Y 240.879,Z 346.889,A -85,B 0,C 180,E1 -19863.346,E2 -19863.346} C_VEL
LIN {X 0,Y 237.46,Z 356.989,A -85,B 0,C 180,E1 -19865.52,E2 -19865.52} C_VEL
LIN {X 0,Y 234.397,Z 365.906,A -85,B 0,C 180,E1 -19867.987,E2 -19867.987} C_VEL
LIN {X 0,Y 231.837,Z 373.135,A -85,B 0,C 180,E1 -19870.52,E2 -19870.52} C_VEL
LIN {X 0,Y 229.713,Z 378.972,A -85,B 0,C 180,E1 -19873.102,E2 -19873.102} C_VEL
LIN {X 0,Y 227.892,Z 383.611,A -85,B 0,C 180,E1 -19875.716,E2 -19875.716} C_VEL
LIN {X 0,Y 226.759,Z 387.18,A -85,B 0,C 180,E1 -19878.377,E2 -19878.377} C_VEL
LIN {X 0,Y 226.035,Z 389.76,A -85,B 0,C 180,E1 -19881.055,E2 -19881.055} C_VEL
LIN {X 0,Y 225.766,Z 390.953,A -85,B 0,C 180,E1 -19882.846,E2 -19882.846} C_VEL
LIN {X 0,Y 225.659,Z 392.141,A -85,B 0,C 180,E1 -19886.428,E2 -19886.428} C_VEL
LIN {X 0,Y 225.8,Z 392.154,A -85,B 0,C 180,E1 -19888.215,E2 -19888.215} C_VEL
LIN {X 0,Y 225.877,Z 391.732,A -85,B 0,C 180,E1 -19889.999,E2 -19889.999} C_VEL
LIN {X 0,Y 225.847,Z 390.869,A -85,B 0,C 180,E1 -19891.782,E2 -19891.782} C_VEL
LIN {X 0,Y 225.747,Z 388.273,A -85,B 0,C 180,E1 -19894.968,E2 -19894.968} C_VEL
LIN {X 0,Y 225.958,Z 384.403,A -85,B 0,C 180,E1 -19898.045,E2 -19898.045} C_VEL
LIN {X 0,Y 226.417,Z 379.782,A -85,B 0,C 180,E1 -19900.732,E2 -19900.732} C_VEL
LIN {X 0,Y 227.442,Z 372.729,A -85,B 0,C 180,E1 -19903.855,E2 -19903.855} C_VEL
LIN {X 0,Y 228.833,Z 365.072,A -85,B 0,C 180,E1 -19906.503,E2 -19906.503} C_VEL
LIN {X 0,Y 230.279,Z 356.856,A -85,B 0,C 180,E1 -19908.784,E2 -19908.784} C_VEL
LIN {X 0,Y 232.259,Z 346.541,A -85,B 0,C 180,E1 -19911.058,E2 -19911.058} C_VEL
LIN {X 0,Y 234.221,Z 335.689,A -85,B 0,C 180,E1 -19912.958,E2 -19912.958} C_VEL
LIN {X 0,Y 235.951,Z 325.156,A -85,B 0,C 180,E1 -19914.41,E2 -19914.41} C_VEL
LIN {X 0,Y 237.704,Z 312.565,A -85,B 0,C 180,E1 -19915.737,E2 -19915.737} C_VEL
LIN {X 0,Y 239.116,Z 299.412,A -85,B 0,C 180,E1 -19916.746,E2 -19916.746} C_VEL
LIN {X 0,Y 240.116,Z 286.315,A -85,B 0,C 180,E1 -19917.391,E2 -19917.391} C_VEL
LIN {X 0,Y 242.054,Z 233.674,A -85,B 0,C 180,E1 -19919.1,E2 -19919.1} C_VEL
LIN {X 0,Y 237.42,Z 197.122,A -85,B 0,C 180,E1 -19920.918,E2 -19920.918} C_VEL
LIN {X 0,Y 231.139,Z 179.827,A -85,B 0,C 180,E1 -19922.326,E2 -19922.326} C_VEL
LIN {X 0,Y 229.065,Z 169.934,A -85,B 0,C 180,E1 -19926.271,E2 -19926.271} C_VEL
LIN {X 0,Y 227.918,Z 165.096,A -85,B 0,C 180,E1 -19928.341,E2 -19928.341} C_VEL
LIN {X 0,Y 227.811,Z 165.111,A -85,B 0,C 180,E1 -19932.741,E2 -19932.741} C_VEL
LIN {X 0,Y 227.811,Z 165.108,A -85,B 0,C 180,E1 -19937.256,E2 -19937.256} C_VEL
LIN {X 0,Y 227.844,Z 165.105,A -85,B 0,C 180,E1 -19941.908,E2 -19941.908} C_VEL
LIN {X 0,Y 227.882,Z 165.098,A -85,B 0,C 180,E1 -19946.375,E2 -19946.375} C_VEL
LIN {X 0,Y 227.919,Z 165.088,A -85,B 0,C 180,E1 -19950.437,E2 -19950.437} C_VEL
LIN {X 0,Y 227.928,Z 165.091,A -85,B 0,C 180,E1 -19954.425,E2 -19954.425} C_VEL
LIN {X 0,Y 227.959,Z 165.087,A -85,B 0,C 180,E1 -19958.286,E2 -19958.286} C_VEL
LIN {X 0,Y 228.021,Z 165.074,A -85,B 0,C 180,E1 -19963.894,E2 -19963.894} C_VEL
LIN {X 0,Y 228.067,Z 165.076,A -85,B 0,C 180,E1 -19967.542,E2 -19967.542} C_VEL
LIN {X 0,Y 228.303,Z 165.039,A -85,B 0,C 180,E1 -19971.145,E2 -19971.145} C_VEL
LIN {X 0,Y 228.352,Z 165.032,A -85,B 0,C 180,E1 -19972.928,E2 -19972.928} C_VEL
LIN {X 0,Y 228.553,Z 165.013,A -85,B 0,C 180,E1 -19978.237,E2 -19978.237} C_VEL
LIN {X 0,Y 228.552,Z 165.004,A -85,B 0,C 180,E1 -19981.761,E2 -19981.761} C_VEL
LIN {X 0,Y 228.351,Z 165.04,A -85,B 0,C 180,E1 -19987.071,E2 -19987.071} C_VEL
LIN {X 0,Y 228.16,Z 165.061,A -85,B 0,C 180,E1 -19990.649,E2 -19990.649} C_VEL
LIN {X 0,Y 228.061,Z 165.063,A -85,B 0,C 180,E1 -19994.271,E2 -19994.271} C_VEL
LIN {X 0,Y 228,Z 165.081,A -85,B 0,C 180,E1 -19997.952,E2 -19997.952} C_VEL
LIN {X 0,Y 227.95,Z 165.087,A -85,B 0,C 180,E1 -20002.343,E2 -20002.343} C_VEL
LIN {X 0,Y 227.939,Z 165.081,A -85,B 0,C 180,E1 -20006.602,E2 -20006.602} C_VEL
LIN {X 0,Y 227.904,Z 165.095,A -85,B 0,C 180,E1 -20010.296,E2 -20010.296} C_VEL
LIN {X 0,Y 227.886,Z 165.093,A -85,B 0,C 180,E1 -20013.718,E2 -20013.718} C_VEL
LIN {X 0,Y 227.886,Z 165.09,A -85,B 0,C 180,E1 -20018.081,E2 -20018.081} C_VEL
LIN {X 0,Y 227.932,Z 165.088,A -85,B 0,C 180,E1 -20022.713,E2 -20022.713} C_VEL
LIN {X 0,Y 227.932,Z 165.084,A -85,B 0,C 180,E1 -20027.287,E2 -20027.287} C_VEL
LIN {X 0,Y 227.886,Z 165.097,A -85,B 0,C 180,E1 -20031.918,E2 -20031.918} C_VEL
LIN {X 0,Y 227.886,Z 165.096,A -85,B 0,C 180,E1 -20036.373,E2 -20036.373} C_VEL
LIN {X 0,Y 227.914,Z 165.092,A -85,B 0,C 180,E1 -20040.438,E2 -20040.438} C_VEL
LIN {X 0,Y 227.924,Z 165.092,A -85,B 0,C 180,E1 -20044.426,E2 -20044.426} C_VEL
LIN {X 0,Y 227.958,Z 165.089,A -85,B 0,C 180,E1 -20048.288,E2 -20048.288} C_VEL
LIN {X 0,Y 228.03,Z 165.08,A -85,B 0,C 180,E1 -20052.826,E2 -20052.826} C_VEL
LIN {X 0,Y 228.09,Z 165.076,A -85,B 0,C 180,E1 -20057.545,E2 -20057.545} C_VEL
LIN {X 0,Y 228.322,Z 165.049,A -85,B 0,C 180,E1 -20061.148,E2 -20061.148} C_VEL
LIN {X 0,Y 228.355,Z 165.043,A -85,B 0,C 180,E1 -20062.93,E2 -20062.93} C_VEL
LIN {X 0,Y 228.552,Z 165.015,A -85,B 0,C 180,E1 -20068.239,E2 -20068.239} C_VEL
LIN {X 0,Y 228.552,Z 165.015,A -85,B 0,C 180,E1 -20071.763,E2 -20071.763} C_VEL
LIN {X 0,Y 228.231,Z 165.089,A -85,B 0,C 180,E1 -20075.634,E2 -20075.634} C_VEL
LIN {X 0,Y 229.275,Z 167.931,A -85,B 0,C 180,E1 -20075.872,E2 -20075.872} C_VEL
LIN {X 0,Y 235.321,Z 180.946,A -85,B 0,C 180,E1 -20077.072,E2 -20077.072} C_VEL
LIN {X 0,Y 241.095,Z 195.506,A -85,B 0,C 180,E1 -20078.236,E2 -20078.236} C_VEL
LIN {X 0,Y 243.157,Z 201.461,A -85,B 0,C 180,E1 -20078.668,E2 -20078.668} C_VEL
LIN {X 0,Y 240.338,Z 268.859,A -85,B 0,C 180,E1 -20080.851,E2 -20080.851} C_VEL
LIN {X 0,Y 239.358,Z 281.851,A -85,B 0,C 180,E1 -20081.593,E2 -20081.593} C_VEL
LIN {X 0,Y 238.219,Z 294.479,A -85,B 0,C 180,E1 -20082.658,E2 -20082.658} C_VEL
LIN {X 0,Y 236.826,Z 305.915,A -85,B 0,C 180,E1 -20083.953,E2 -20083.953} C_VEL
LIN {X 0,Y 235.001,Z 317.422,A -85,B 0,C 180,E1 -20085.615,E2 -20085.615} C_VEL
LIN {X 0,Y 233.142,Z 327.989,A -85,B 0,C 180,E1 -20087.546,E2 -20087.546} C_VEL
LIN {X 0,Y 231.45,Z 337.446,A -85,B 0,C 180,E1 -20089.729,E2 -20089.729} C_VEL
LIN {X 0,Y 229.911,Z 345.418,A -85,B 0,C 180,E1 -20091.992,E2 -20091.992} C_VEL
LIN {X 0,Y 228.538,Z 352.649,A -85,B 0,C 180,E1 -20094.53,E2 -20094.53} C_VEL
LIN {X 0,Y 227.499,Z 358.282,A -85,B 0,C 180,E1 -20096.994,E2 -20096.994} C_VEL
LIN {X 0,Y 226.664,Z 363.269,A -85,B 0,C 180,E1 -20099.755,E2 -20099.755} C_VEL
LIN {X 0,Y 225.945,Z 367.424,A -85,B 0,C 180,E1 -20102.88,E2 -20102.88} C_VEL
LIN {X 0,Y 225.481,Z 370.396,A -85,B 0,C 180,E1 -20106.315,E2 -20106.315} C_VEL
LIN {X 0,Y 225.502,Z 371.592,A -85,B 0,C 180,E1 -20108.819,E2 -20108.819} C_VEL
LIN {X 0,Y 225.795,Z 371.997,A -85,B 0,C 180,E1 -20111.669,E2 -20111.669} C_VEL
LIN {X 0,Y 226.426,Z 371.411,A -85,B 0,C 180,E1 -20114.449,E2 -20114.449} C_VEL
LIN {X 0,Y 227.554,Z 369.368,A -85,B 0,C 180,E1 -20117.839,E2 -20117.839} C_VEL
LIN {X 0,Y 228.729,Z 367.015,A -85,B 0,C 180,E1 -20120.19,E2 -20120.19} C_VEL
LIN {X 0,Y 230.119,Z 363.824,A -85,B 0,C 180,E1 -20122.568,E2 -20122.568} C_VEL
LIN {X 0,Y 232.387,Z 358.528,A -85,B 0,C 180,E1 -20125.5,E2 -20125.5} C_VEL
LIN {X 0,Y 235.198,Z 351.638,A -85,B 0,C 180,E1 -20128.388,E2 -20128.388} C_VEL
LIN {X 0,Y 237.798,Z 344.63,A -85,B 0,C 180,E1 -20130.675,E2 -20130.675} C_VEL
LIN {X 0,Y 240.813,Z 335.944,A -85,B 0,C 180,E1 -20132.923,E2 -20132.923} C_VEL
LIN {X 0,Y 243.718,Z 326.51,A -85,B 0,C 180,E1 -20134.878,E2 -20134.878} C_VEL
LIN {X 0,Y 246.67,Z 315.841,A -85,B 0,C 180,E1 -20136.618,E2 -20136.618} C_VEL
LIN {X 0,Y 249.176,Z 304.768,A -85,B 0,C 180,E1 -20138.035,E2 -20138.035} C_VEL
LIN {X 0,Y 251.335,Z 292.798,A -85,B 0,C 180,E1 -20139.222,E2 -20139.222} C_VEL
LIN {X 0,Y 253.052,Z 280.149,A -85,B 0,C 180,E1 -20140.149,E2 -20140.149} C_VEL
LIN {X 0,Y 254.2,Z 268.139,A -85,B 0,C 180,E1 -20140.728,E2 -20140.728} C_VEL
LIN {X 0,Y 257.411,Z 213.534,A -85,B 0,C 180,E1 -20142.455,E2 -20142.455} C_VEL
LIN {X 0,Y 251.442,Z 200.916,A -85,B 0,C 180,E1 -20144.322,E2 -20144.322} C_VEL
LIN {X 0,Y 246.195,Z 191.35,A -85,B 0,C 180,E1 -20146.072,E2 -20146.072} C_VEL
LIN {X 0,Y 240.911,Z 183.38,A -85,B 0,C 180,E1 -20147.909,E2 -20147.909} C_VEL
LIN {X 0,Y 237.892,Z 179.098,A -85,B 0,C 180,E1 -20149.038,E2 -20149.038} C_VEL
LIN {X 0,Y 235.156,Z 175.12,A -85,B 0,C 180,E1 -20150.126,E2 -20150.126} C_VEL
LIN {X 0,Y 232.955,Z 172.414,A -85,B 0,C 180,E1 -20151.023,E2 -20151.023} C_VEL
LIN {X 0,Y 231.924,Z 170.39,A -85,B 0,C 180,E1 -20151.506,E2 -20151.506} C_VEL
LIN {X 0,Y 229.733,Z 168.563,A -85,B 0,C 180,E1 -20152.42,E2 -20152.42} C_VEL
LIN {X 0,Y 228.52,Z 166.08,A -85,B 0,C 180,E1 -20153.046,E2 -20153.046} C_VEL
LIN {X 0,Y 228.304,Z 165.046,A -85,B 0,C 180,E1 -20153.261,E2 -20153.261} C_VEL
LIN {X 0,Y 228.539,Z 165.012,A -85,B 0,C 180,E1 -20158.239,E2 -20158.239} C_VEL
LIN {X 0,Y 228.537,Z 165.012,A -85,B 0,C 180,E1 -20161.763,E2 -20161.763} C_VEL
LIN {X 0,Y 228.304,Z 165.032,A -85,B 0,C 180,E1 -20167.074,E2 -20167.074} C_VEL
LIN {X 0,Y 228.129,Z 165.053,A -85,B 0,C 180,E1 -20170.653,E2 -20170.653} C_VEL
LIN {X 0,Y 228.003,Z 165.072,A -85,B 0,C 180,E1 -20176.107,E2 -20176.107} C_VEL
LIN {X 0,Y 227.872,Z 165.089,A -85,B 0,C 180,E1 -20180.506,E2 -20180.506} C_VEL
LIN {X 0,Y 227.205,Z 165.183,A -85,B 0,C 180,E1 -20181.98,E2 -20181.98} C_VEL
LIN {X 0,Y 224.34,Z 165.53,A -85,B 0,C 180,E1 -20184.385,E2 -20184.385} C_VEL
LIN {X 0,Y 221.909,Z 165.839,A -85,B 0,C 180,E1 -20186.347,E2 -20186.347} C_VEL
LIN {X 0,Y 220.877,Z 165.96,A -85,B 0,C 180,E1 -20187.872,E2 -20187.872} C_VEL
LIN {X 0,Y 220.799,Z 165.971,A -85,B 0,C 180,E1 -20188.388,E2 -20188.388} C_VEL
LIN {X 0,Y 220.817,Z 165.974,A -85,B 0,C 180,E1 -20192.757,E2 -20192.757} C_VEL
LIN {X 0,Y 220.852,Z 166.047,A -85,B 0,C 180,E1 -20195.645,E2 -20195.645} C_VEL
LIN {X 0,Y 222.118,Z 170.083,A -85,B 0,C 180,E1 -20199.259,E2 -20199.259} C_VEL
LIN {X 0,Y 223.762,Z 174.969,A -85,B 0,C 180,E1 -20202.992,E2 -20202.992} C_VEL
LIN {X 0,Y 226.903,Z 179.858,A -85,B 0,C 180,E1 -20204.587,E2 -20204.587} C_VEL
LIN {X 0,Y 228.61,Z 182.198,A -85,B 0,C 180,E1 -20205.383,E2 -20205.383} C_VEL
LIN {X 0,Y 232.604,Z 188.553,A -85,B 0,C 180,E1 -20207.167,E2 -20207.167} C_VEL
LIN {X 0,Y 236.463,Z 195.089,A -85,B 0,C 180,E1 -20208.759,E2 -20208.759} C_VEL
LIN {X 0,Y 240.749,Z 202.884,A -85,B 0,C 180,E1 -20210.416,E2 -20210.416} C_VEL
LIN {X 0,Y 246.242,Z 214.516,A -85,B 0,C 180,E1 -20212.415,E2 -20212.415} C_VEL
LIN {X 0,Y 249.052,Z 221.642,A -85,B 0,C 180,E1 -20213.426,E2 -20213.426} C_VEL
LIN {X 0,Y 250.777,Z 237.658,A -85,B 0,C 180,E1 -20214.536,E2 -20214.536} C_VEL
LIN {X 0,Y 250.876,Z 241.202,A -85,B 0,C 180,E1 -20214.717,E2 -20214.717} C_VEL
LIN {X 0,Y 247.87,Z 287.546,A -85,B 0,C 180,E1 -20216.215,E2 -20216.215} C_VEL
LIN {X 0,Y 246.178,Z 300.935,A -85,B 0,C 180,E1 -20216.923,E2 -20216.923} C_VEL
LIN {X 0,Y 243.989,Z 312.701,A -85,B 0,C 180,E1 -20217.798,E2 -20217.798} C_VEL
LIN {X 0,Y 241.17,Z 325.153,A -85,B 0,C 180,E1 -20219.094,E2 -20219.094} C_VEL
LIN {X 0,Y 238.025,Z 336.36,A -85,B 0,C 180,E1 -20220.601,E2 -20220.601} C_VEL
LIN {X 0,Y 234.927,Z 346.586,A -85,B 0,C 180,E1 -20222.373,E2 -20222.373} C_VEL
LIN {X 0,Y 231.692,Z 355.858,A -85,B 0,C 180,E1 -20224.388,E2 -20224.388} C_VEL
LIN {X 0,Y 228.316,Z 364.913,A -85,B 0,C 180,E1 -20226.891,E2 -20226.891} C_VEL
LIN {X 0,Y 225.601,Z 372.292,A -85,B 0,C 180,E1 -20229.499,E2 -20229.499} C_VEL
LIN {X 0,Y 223.583,Z 377.266,A -85,B 0,C 180,E1 -20231.678,E2 -20231.678} C_VEL
LIN {X 0,Y 221.606,Z 382.177,A -85,B 0,C 180,E1 -20234.36,E2 -20234.36} C_VEL
LIN {X 0,Y 220.107,Z 385.999,A -85,B 0,C 180,E1 -20237.084,E2 -20237.084} C_VEL
LIN {X 0,Y 219.473,Z 388.005,A -85,B 0,C 180,E1 -20238.922,E2 -20238.922} C_VEL
LIN {X 0,Y 219.001,Z 389.58,A -85,B 0,C 180,E1 -20240.766,E2 -20240.766} C_VEL
LIN {X 0,Y 218.567,Z 391.467,A -85,B 0,C 180,E1 -20244.463,E2 -20244.463} C_VEL
LIN {X 0,Y 218.567,Z 391.83,A -85,B 0,C 180,E1 -20246.312,E2 -20246.312} C_VEL
LIN {X 0,Y 218.706,Z 391.794,A -85,B 0,C 180,E1 -20248.157,E2 -20248.157} C_VEL
LIN {X 0,Y 218.808,Z 391.311,A -85,B 0,C 180,E1 -20249.999,E2 -20249.999} C_VEL
LIN {X 0,Y 218.777,Z 390.412,A -85,B 0,C 180,E1 -20251.84,E2 -20251.84} C_VEL
LIN {X 0,Y 218.655,Z 388.011,A -85,B 0,C 180,E1 -20254.851,E2 -20254.851} C_VEL
LIN {X 0,Y 218.806,Z 385.056,A -85,B 0,C 180,E1 -20257.381,E2 -20257.381} C_VEL
LIN {X 0,Y 219.214,Z 380.743,A -85,B 0,C 180,E1 -20260.155,E2 -20260.155} C_VEL
LIN {X 0,Y 220.117,Z 374.157,A -85,B 0,C 180,E1 -20263.383,E2 -20263.383} C_VEL
LIN {X 0,Y 221.461,Z 366.893,A -85,B 0,C 180,E1 -20266.121,E2 -20266.121} C_VEL
LIN {X 0,Y 222.846,Z 359.475,A -85,B 0,C 180,E1 -20268.382,E2 -20268.382} C_VEL
LIN {X 0,Y 224.582,Z 350.48,A -85,B 0,C 180,E1 -20270.612,E2 -20270.612} C_VEL
LIN {X 0,Y 226.488,Z 340.617,A -85,B 0,C 180,E1 -20272.581,E2 -20272.581} C_VEL
LIN {X 0,Y 228.433,Z 329.803,A -85,B 0,C 180,E1 -20274.298,E2 -20274.298} C_VEL
LIN {X 0,Y 230.231,Z 317.697,A -85,B 0,C 180,E1 -20275.784,E2 -20275.784} C_VEL
LIN {X 0,Y 231.885,Z 305.24,A -85,B 0,C 180,E1 -20276.918,E2 -20276.918} C_VEL
LIN {X 0,Y 233.09,Z 292.287,A -85,B 0,C 180,E1 -20277.739,E2 -20277.739} C_VEL
LIN {X 0,Y 234.006,Z 274.443,A -85,B 0,C 180,E1 -20278.413,E2 -20278.413} C_VEL
LIN {X 0,Y 235.487,Z 234.268,A -85,B 0,C 180,E1 -20279.745,E2 -20279.745} C_VEL
LIN {X 0,Y 231.093,Z 199.228,A -85,B 0,C 180,E1 -20281.534,E2 -20281.534} C_VEL
LIN {X 0,Y 223.817,Z 179.491,A -85,B 0,C 180,E1 -20283.22,E2 -20283.22} C_VEL
LIN {X 0,Y 221.609,Z 169.1,A -85,B 0,C 180,E1 -20287.547,E2 -20287.547} C_VEL
LIN {X 0,Y 220.856,Z 165.975,A -85,B 0,C 180,E1 -20288.984,E2 -20288.984} C_VEL
LIN {X 0,Y 220.766,Z 165.989,A -85,B 0,C 180,E1 -20292.928,E2 -20292.928} C_VEL
LIN {X 0,Y 220.766,Z 165.985,A -85,B 0,C 180,E1 -20297.069,E2 -20297.069} C_VEL
LIN {X 0,Y 220.806,Z 165.98,A -85,B 0,C 180,E1 -20300.462,E2 -20300.462} C_VEL
LIN {X 0,Y 220.803,Z 165.981,A -85,B 0,C 180,E1 -20305.044,E2 -20305.044} C_VEL
LIN {X 0,Y 220.867,Z 165.971,A -85,B 0,C 180,E1 -20309.394,E2 -20309.394} C_VEL
LIN {X 0,Y 220.895,Z 165.97,A -85,B 0,C 180,E1 -20313.548,E2 -20313.548} C_VEL
LIN {X 0,Y 220.877,Z 165.97,A -85,B 0,C 180,E1 -20317.552,E2 -20317.552} C_VEL
LIN {X 0,Y 220.928,Z 165.961,A -85,B 0,C 180,E1 -20322.615,E2 -20322.615} C_VEL
LIN {X 0,Y 221.003,Z 165.958,A -85,B 0,C 180,E1 -20327.137,E2 -20327.137} C_VEL
LIN {X 0,Y 221.234,Z 165.921,A -85,B 0,C 180,E1 -20330.86,E2 -20330.86} C_VEL
LIN {X 0,Y 221.287,Z 165.91,A -85,B 0,C 180,E1 -20332.701,E2 -20332.701} C_VEL
LIN {X 0,Y 221.511,Z 165.891,A -85,B 0,C 180,E1 -20338.181,E2 -20338.181} C_VEL
LIN {X 0,Y 221.51,Z 165.88,A -85,B 0,C 180,E1 -20341.817,E2 -20341.817} C_VEL
LIN {X 0,Y 221.286,Z 165.919,A -85,B 0,C 180,E1 -20347.298,E2 -20347.298} C_VEL
LIN {X 0,Y 221.109,Z 165.937,A -85,B 0,C 180,E1 -20350.993,E2 -20350.993} C_VEL
LIN {X 0,Y 221.013,Z 165.95,A -85,B 0,C 180,E1 -20356.629,E2 -20356.629} C_VEL
LIN {X 0,Y 220.896,Z 165.969,A -85,B 0,C 180,E1 -20360.485,E2 -20360.485} C_VEL
LIN {X 0,Y 220.868,Z 165.958,A -85,B 0,C 180,E1 -20364.434,E2 -20364.434} C_VEL
LIN {X 0,Y 220.833,Z 165.972,A -85,B 0,C 180,E1 -20368.513,E2 -20368.513} C_VEL
LIN {X 0,Y 220.82,Z 165.973,A -85,B 0,C 180,E1 -20372.754,E2 -20372.754} C_VEL
LIN {X 0,Y 220.863,Z 165.96,A -85,B 0,C 180,E1 -20377.298,E2 -20377.298} C_VEL
LIN {X 0,Y 220.875,Z 165.971,A -85,B 0,C 180,E1 -20381.927,E2 -20381.927} C_VEL
LIN {X 0,Y 220.87,Z 165.963,A -85,B 0,C 180,E1 -20385.572,E2 -20385.572} C_VEL
LIN {X 0,Y 220.873,Z 165.972,A -85,B 0,C 180,E1 -20389.786,E2 -20389.786} C_VEL
LIN {X 0,Y 220.839,Z 165.972,A -85,B 0,C 180,E1 -20392.797,E2 -20392.797} C_VEL
LIN {X 0,Y 220.82,Z 165.977,A -85,B 0,C 180,E1 -20397.246,E2 -20397.246} C_VEL
LIN {X 0,Y 220.832,Z 165.978,A -85,B 0,C 180,E1 -20401.487,E2 -20401.487} C_VEL
LIN {X 0,Y 220.863,Z 165.975,A -85,B 0,C 180,E1 -20405.566,E2 -20405.566} C_VEL
LIN {X 0,Y 220.888,Z 165.971,A -85,B 0,C 180,E1 -20409.515,E2 -20409.515} C_VEL
LIN {X 0,Y 221.012,Z 165.957,A -85,B 0,C 180,E1 -20413.371,E2 -20413.371} C_VEL
LIN {X 0,Y 221.113,Z 165.946,A -85,B 0,C 180,E1 -20419.007,E2 -20419.007} C_VEL
LIN {X 0,Y 221.308,Z 165.92,A -85,B 0,C 180,E1 -20422.703,E2 -20422.703} C_VEL
LIN {X 0,Y 221.51,Z 165.893,A -85,B 0,C 180,E1 -20428.183,E2 -20428.183} C_VEL
LIN {X 0,Y 221.51,Z 165.892,A -85,B 0,C 180,E1 -20431.819,E2 -20431.819} C_VEL
LIN {X 0,Y 221.17,Z 166.09,A -85,B 0,C 180,E1 -20434.786,E2 -20434.786} C_VEL
LIN {X 0,Y 222.196,Z 168.834,A -85,B 0,C 180,E1 -20435.029,E2 -20435.029} C_VEL
LIN {X 0,Y 228.705,Z 182.39,A -85,B 0,C 180,E1 -20436.368,E2 -20436.368} C_VEL
LIN {X 0,Y 234.942,Z 198.163,A -85,B 0,C 180,E1 -20437.676,E2 -20437.676} C_VEL
LIN {X 0,Y 236.581,Z 202.911,A -85,B 0,C 180,E1 -20438.028,E2 -20438.028} C_VEL
LIN {X 0,Y 233.741,Z 268.99,A -85,B 0,C 180,E1 -20440.23,E2 -20440.23} C_VEL
LIN {X 0,Y 232.726,Z 282.024,A -85,B 0,C 180,E1 -20440.991,E2 -20440.991} C_VEL
LIN {X 0,Y 231.601,Z 294.267,A -85,B 0,C 180,E1 -20442.043,E2 -20442.043} C_VEL
LIN {X 0,Y 230.058,Z 306.383,A -85,B 0,C 180,E1 -20443.444,E2 -20443.444} C_VEL
LIN {X 0,Y 228.139,Z 318.04,A -85,B 0,C 180,E1 -20445.181,E2 -20445.181} C_VEL
LIN {X 0,Y 226.245,Z 328.565,A -85,B 0,C 180,E1 -20447.174,E2 -20447.174} C_VEL
LIN {X 0,Y 224.383,Z 338.338,A -85,B 0,C 180,E1 -20449.516,E2 -20449.516} C_VEL
LIN {X 0,Y 222.609,Z 347.474,A -85,B 0,C 180,E1 -20452.264,E2 -20452.264} C_VEL
LIN {X 0,Y 221.236,Z 354.373,A -85,B 0,C 180,E1 -20454.893,E2 -20454.893} C_VEL
LIN {X 0,Y 220.145,Z 360.133,A -85,B 0,C 180,E1 -20457.657,E2 -20457.657} C_VEL
LIN {X 0,Y 219.272,Z 365.231,A -85,B 0,C 180,E1 -20460.853,E2 -20460.853} C_VEL
LIN {X 0,Y 218.74,Z 368.175,A -85,B 0,C 180,E1 -20463.348,E2 -20463.348} C_VEL
LIN {X 0,Y 218.403,Z 370.704,A -85,B 0,C 180,E1 -20466.442,E2 -20466.442} C_VEL
LIN {X 0,Y 218.498,Z 372.197,A -85,B 0,C 180,E1 -20470.04,E2 -20470.04} C_VEL
LIN {X 0,Y 218.847,Z 372.315,A -85,B 0,C 180,E1 -20472.408,E2 -20472.408} C_VEL
LIN {X 0,Y 219.522,Z 371.612,A -85,B 0,C 180,E1 -20475.226,E2 -20475.226} C_VEL
LIN {X 0,Y 220.512,Z 369.996,A -85,B 0,C 180,E1 -20477.989,E2 -20477.989} C_VEL
LIN {X 0,Y 221.901,Z 367.466,A -85,B 0,C 180,E1 -20480.697,E2 -20480.697} C_VEL
LIN {X 0,Y 223.491,Z 364.072,A -85,B 0,C 180,E1 -20483.312,E2 -20483.312} C_VEL
LIN {X 0,Y 225.931,Z 358.76,A -85,B 0,C 180,E1 -20486.324,E2 -20486.324} C_VEL
LIN {X 0,Y 228.921,Z 351.842,A -85,B 0,C 180,E1 -20489.275,E2 -20489.275} C_VEL
LIN {X 0,Y 231.69,Z 344.812,A -85,B 0,C 180,E1 -20491.605,E2 -20491.605} C_VEL
LIN {X 0,Y 234.825,Z 336.173,A -85,B 0,C 180,E1 -20493.88,E2 -20493.88} C_VEL
LIN {X 0,Y 237.948,Z 326.605,A -85,B 0,C 180,E1 -20495.889,E2 -20495.889} C_VEL
LIN {X 0,Y 240.817,Z 316.729,A -85,B 0,C 180,E1 -20497.539,E2 -20497.539} C_VEL
LIN {X 0,Y 243.397,Z 306.114,A -85,B 0,C 180,E1 -20498.948,E2 -20498.948} C_VEL
LIN {X 0,Y 245.703,Z 294.173,A -85,B 0,C 180,E1 -20500.179,E2 -20500.179} C_VEL
LIN {X 0,Y 247.471,Z 282.159,A -85,B 0,C 180,E1 -20501.101,E2 -20501.101} C_VEL
LIN {X 0,Y 248.731,Z 270.407,A -85,B 0,C 180,E1 -20501.72,E2 -20501.72} C_VEL
LIN {X 0,Y 252.135,Z 215.927,A -85,B 0,C 180,E1 -20503.48,E2 -20503.48} C_VEL
LIN {X 0,Y 246.806,Z 204.666,A -85,B 0,C 180,E1 -20505.264,E2 -20505.264} C_VEL
LIN {X 0,Y 242.25,Z 196.251,A -85,B 0,C 180,E1 -20506.856,E2 -20506.856} C_VEL
LIN {X 0,Y 237.396,Z 188.757,A -85,B 0,C 180,E1 -20508.65,E2 -20508.65} C_VEL
LIN {X 0,Y 234.571,Z 184.675,A -85,B 0,C 180,E1 -20509.754,E2 -20509.754} C_VEL
LIN {X 0,Y 231.833,Z 180.718,A -85,B 0,C 180,E1 -20510.898,E2 -20510.898} C_VEL
LIN {X 0,Y 229.432,Z 177.292,A -85,B 0,C 180,E1 -20511.967,E2 -20511.967} C_VEL
LIN {X 0,Y 228.756,Z 176.355,A -85,B 0,C 180,E1 -20512.276,E2 -20512.276} C_VEL
LIN {X 0,Y 226.351,Z 173.65,A -85,B 0,C 180,E1 -20513.38,E2 -20513.38} C_VEL
LIN {X 0,Y 225.367,Z 171.576,A -85,B 0,C 180,E1 -20513.916,E2 -20513.916} C_VEL
LIN {X 0,Y 222.827,Z 169.722,A -85,B 0,C 180,E1 -20515.139,E2 -20515.139} C_VEL
LIN {X 0,Y 221.501,Z 167.483,A -85,B 0,C 180,E1 -20515.907,E2 -20515.907} C_VEL
LIN {X 0,Y 221.149,Z 165.932,A -85,B 0,C 180,E1 -20516.243,E2 -20516.243} C_VEL
LIN {X 0,Y 221.473,Z 165.892,A -85,B 0,C 180,E1 -20518.183,E2 -20518.183} C_VEL
LIN {X 0,Y 221.47,Z 165.891,A -85,B 0,C 180,E1 -20521.819,E2 -20521.819} C_VEL
LIN {X 0,Y 221.241,Z 165.912,A -85,B 0,C 180,E1 -20527.301,E2 -20527.301} C_VEL
LIN {X 0,Y 221.054,Z 165.934,A -85,B 0,C 180,E1 -20530.998,E2 -20530.998} C_VEL
LIN {X 0,Y 220.97,Z 165.952,A -85,B 0,C 180,E1 -20536.634,E2 -20536.634} C_VEL
LIN {X 0,Y 220.848,Z 165.965,A -85,B 0,C 180,E1 -20540.491,E2 -20540.491} C_VEL
LIN {X 0,Y 220.8,Z 165.97,A -85,B 0,C 180,E1 -20544.444,E2 -20544.444} C_VEL
LIN {X 0,Y 220.799,Z 165.971,A -85,B 0,C 180,E1 -20548.388,E2 -20548.388} C_VEL
LIN {X 0,Y 220.21,Z 166.189,A -85,B 0,C 180,E1 -20549.909,E2 -20549.909} C_VEL
LIN {X 0,Y 217.705,Z 167.351,A -85,B 0,C 180,E1 -20552.393,E2 -20552.393} C_VEL
LIN {X 0,Y 215.72,Z 168.887,A -85,B 0,C 180,E1 -20554.396,E2 -20554.396} C_VEL
LIN {X 0,Y 215.073,Z 170.332,A -85,B 0,C 180,E1 -20555.922,E2 -20555.922} C_VEL
LIN {X 0,Y 215.128,Z 170.861,A -85,B 0,C 180,E1 -20556.43,E2 -20556.43} C_VEL
LIN {X 0,Y 216.195,Z 174.082,A -85,B 0,C 180,E1 -20559.338,E2 -20559.338} C_VEL
LIN {X 0,Y 219.639,Z 179.313,A -85,B 0,C 180,E1 -20561.478,E2 -20561.478} C_VEL
LIN {X 0,Y 221.347,Z 181.472,A -85,B 0,C 180,E1 -20562.418,E2 -20562.418} C_VEL
LIN {X 0,Y 224.927,Z 186.785,A -85,B 0,C 180,E1 -20564.286,E2 -20564.286} C_VEL
LIN {X 0,Y 229.719,Z 194.731,A -85,B 0,C 180,E1 -20566.57,E2 -20566.57} C_VEL
LIN {X 0,Y 233.25,Z 200.897,A -85,B 0,C 180,E1 -20568.097,E2 -20568.097} C_VEL
LIN {X 0,Y 237.171,Z 208.33,A -85,B 0,C 180,E1 -20569.699,E2 -20569.699} C_VEL
LIN {X 0,Y 242.25,Z 219.47,A -85,B 0,C 180,E1 -20571.654,E2 -20571.654} C_VEL
LIN {X 0,Y 244.271,Z 224.842,A -85,B 0,C 180,E1 -20572.431,E2 -20572.431} C_VEL
LIN {X 0,Y 245.784,Z 240.889,A -85,B 0,C 180,E1 -20573.574,E2 -20573.574} C_VEL
LIN {X 0,Y 242.722,Z 286.419,A -85,B 0,C 180,E1 -20575.056,E2 -20575.056} C_VEL
LIN {X 0,Y 240.925,Z 300.162,A -85,B 0,C 180,E1 -20575.773,E2 -20575.773} C_VEL
LIN {X 0,Y 238.534,Z 312.696,A -85,B 0,C 180,E1 -20576.717,E2 -20576.717} C_VEL
LIN {X 0,Y 235.594,Z 325.063,A -85,B 0,C 180,E1 -20578.027,E2 -20578.027} C_VEL
LIN {X 0,Y 232.292,Z 336.233,A -85,B 0,C 180,E1 -20579.55,E2 -20579.55} C_VEL
LIN {X 0,Y 229.046,Z 346.378,A -85,B 0,C 180,E1 -20581.35,E2 -20581.35} C_VEL
LIN {X 0,Y 225.338,Z 356.4,A -85,B 0,C 180,E1 -20583.611,E2 -20583.611} C_VEL
LIN {X 0,Y 221.83,Z 365.287,A -85,B 0,C 180,E1 -20586.174,E2 -20586.174} C_VEL
LIN {X 0,Y 219.27,Z 371.817,A -85,B 0,C 180,E1 -20588.563,E2 -20588.563} C_VEL
LIN {X 0,Y 216.824,Z 377.412,A -85,B 0,C 180,E1 -20591.086,E2 -20591.086} C_VEL
LIN {X 0,Y 214.775,Z 382.223,A -85,B 0,C 180,E1 -20593.849,E2 -20593.849} C_VEL
LIN {X 0,Y 213.149,Z 385.943,A -85,B 0,C 180,E1 -20596.654,E2 -20596.654} C_VEL
LIN {X 0,Y 212.466,Z 387.892,A -85,B 0,C 180,E1 -20598.551,E2 -20598.551} C_VEL
LIN {X 0,Y 211.982,Z 389.386,A -85,B 0,C 180,E1 -20600.457,E2 -20600.457} C_VEL
LIN {X 0,Y 211.488,Z 391.195,A -85,B 0,C 180,E1 -20604.277,E2 -20604.277} C_VEL
LIN {X 0,Y 211.489,Z 391.519,A -85,B 0,C 180,E1 -20606.188,E2 -20606.188} C_VEL
LIN {X 0,Y 211.614,Z 391.409,A -85,B 0,C 180,E1 -20608.096,E2 -20608.096} C_VEL
LIN {X 0,Y 211.74,Z 390.886,A -85,B 0,C 180,E1 -20609.999,E2 -20609.999} C_VEL
LIN {X 0,Y 211.685,Z 389.947,A -85,B 0,C 180,E1 -20611.901,E2 -20611.901} C_VEL
LIN {X 0,Y 211.565,Z 387.726,A -85,B 0,C 180,E1 -20614.734,E2 -20614.734} C_VEL
LIN {X 0,Y 211.731,Z 384.419,A -85,B 0,C 180,E1 -20617.629,E2 -20617.629} C_VEL
LIN {X 0,Y 212.167,Z 380.01,A -85,B 0,C 180,E1 -20620.496,E2 -20620.496} C_VEL
LIN {X 0,Y 212.96,Z 374.352,A -85,B 0,C 180,E1 -20623.355,E2 -20623.355} C_VEL
LIN {X 0,Y 214.36,Z 367.266,A -85,B 0,C 180,E1 -20626.18,E2 -20626.18} C_VEL
LIN {X 0,Y 215.767,Z 359.987,A -85,B 0,C 180,E1 -20628.515,E2 -20628.515} C_VEL
LIN {X 0,Y 217.491,Z 351.146,A -85,B 0,C 180,E1 -20630.82,E2 -20630.82} C_VEL
LIN {X 0,Y 219.67,Z 340.295,A -85,B 0,C 180,E1 -20633.073,E2 -20633.073} C_VEL
LIN {X 0,Y 221.667,Z 329.476,A -85,B 0,C 180,E1 -20634.839,E2 -20634.839} C_VEL
LIN {X 0,Y 223.524,Z 317.369,A -85,B 0,C 180,E1 -20636.366,E2 -20636.366} C_VEL
LIN {X 0,Y 225.226,Z 304.924,A -85,B 0,C 180,E1 -20637.529,E2 -20637.529} C_VEL
LIN {X 0,Y 226.466,Z 291.991,A -85,B 0,C 180,E1 -20638.371,E2 -20638.371} C_VEL
LIN {X 0,Y 227.422,Z 274.221,A -85,B 0,C 180,E1 -20639.061,E2 -20639.061} C_VEL
LIN {X 0,Y 228.946,Z 235.286,A -85,B 0,C 180,E1 -20640.387,E2 -20640.387} C_VEL
LIN {X 0,Y 224.819,Z 201.428,A -85,B 0,C 180,E1 -20642.169,E2 -20642.169} C_VEL
LIN {X 0,Y 217.511,Z 181.954,A -85,B 0,C 180,E1 -20643.87,E2 -20643.87} C_VEL
LIN {X 0,Y 216.549,Z 179.124,A -85,B 0,C 180,E1 -20644.179,E2 -20644.179} C_VEL
LIN {X 0,Y 214.505,Z 169.944,A -85,B 0,C 180,E1 -20648.154,E2 -20648.154} C_VEL
LIN {X 0,Y 213.788,Z 166.859,A -85,B 0,C 180,E1 -20649.61,E2 -20649.61} C_VEL
LIN {X 0,Y 213.706,Z 166.868,A -85,B 0,C 180,E1 -20653.677,E2 -20653.677} C_VEL
LIN {X 0,Y 213.706,Z 166.865,A -85,B 0,C 180,E1 -20656.343,E2 -20656.343} C_VEL
LIN {X 0,Y 213.717,Z 166.862,A -85,B 0,C 180,E1 -20659.142,E2 -20659.142} C_VEL
LIN {X 0,Y 213.744,Z 166.863,A -85,B 0,C 180,E1 -20663.711,E2 -20663.711} C_VEL
LIN {X 0,Y 213.795,Z 166.854,A -85,B 0,C 180,E1 -20668.723,E2 -20668.723} C_VEL
LIN {X 0,Y 213.825,Z 166.848,A -85,B 0,C 180,E1 -20672.602,E2 -20672.602} C_VEL
LIN {X 0,Y 213.851,Z 166.84,A -85,B 0,C 180,E1 -20676.952,E2 -20676.952} C_VEL
LIN {X 0,Y 213.891,Z 166.837,A -85,B 0,C 180,E1 -20682.798,E2 -20682.798} C_VEL
LIN {X 0,Y 213.941,Z 166.834,A -85,B 0,C 180,E1 -20686.705,E2 -20686.705} C_VEL
LIN {X 0,Y 214.166,Z 166.804,A -85,B 0,C 180,E1 -20690.555,E2 -20690.555} C_VEL
LIN {X 0,Y 214.225,Z 166.789,A -85,B 0,C 180,E1 -20692.458,E2 -20692.458} C_VEL
LIN {X 0,Y 214.444,Z 166.771,A -85,B 0,C 180,E1 -20698.121,E2 -20698.121} C_VEL
LIN {X 0,Y 214.552,Z 166.754,A -85,B 0,C 180,E1 -20699.999,E2 -20699.999} C_VEL
LIN {X 0,Y 214.443,Z 166.76,A -85,B 0,C 180,E1 -20701.877,E2 -20701.877} C_VEL
LIN {X 0,Y 214.224,Z 166.799,A -85,B 0,C 180,E1 -20707.539,E2 -20707.539} C_VEL
LIN {X 0,Y 214.041,Z 166.815,A -85,B 0,C 180,E1 -20711.361,E2 -20711.361} C_VEL
LIN {X 0,Y 213.93,Z 166.827,A -85,B 0,C 180,E1 -20715.236,E2 -20715.236} C_VEL
LIN {X 0,Y 213.838,Z 166.846,A -85,B 0,C 180,E1 -20719.186,E2 -20719.186} C_VEL
LIN {X 0,Y 213.85,Z 166.838,A -85,B 0,C 180,E1 -20723.225,E2 -20723.225} C_VEL
LIN {X 0,Y 213.825,Z 166.839,A -85,B 0,C 180,E1 -20727.449,E2 -20727.449} C_VEL
LIN {X 0,Y 213.775,Z 166.853,A -85,B 0,C 180,E1 -20731.735,E2 -20731.735} C_VEL
LIN {X 0,Y 213.755,Z 166.844,A -85,B 0,C 180,E1 -20736.285,E2 -20736.285} C_VEL
LIN {X 0,Y 213.826,Z 166.846,A -85,B 0,C 180,E1 -20741.097,E2 -20741.097} C_VEL
LIN {X 0,Y 213.831,Z 166.845,A -85,B 0,C 180,E1 -20743.693,E2 -20743.693} C_VEL
LIN {X 0,Y 213.836,Z 166.838,A -85,B 0,C 180,E1 -20746.356,E2 -20746.356} C_VEL
LIN {X 0,Y 213.826,Z 166.846,A -85,B 0,C 180,E1 -20749.107,E2 -20749.107} C_VEL
LIN {X 0,Y 213.755,Z 166.852,A -85,B 0,C 180,E1 -20753.715,E2 -20753.715} C_VEL
LIN {X 0,Y 213.791,Z 166.853,A -85,B 0,C 180,E1 -20758.725,E2 -20758.725} C_VEL
LIN {X 0,Y 213.821,Z 166.849,A -85,B 0,C 180,E1 -20762.604,E2 -20762.604} C_VEL
LIN {X 0,Y 213.848,Z 166.846,A -85,B 0,C 180,E1 -20766.953,E2 -20766.953} C_VEL
LIN {X 0,Y 213.94,Z 166.836,A -85,B 0,C 180,E1 -20772.804,E2 -20772.804} C_VEL
LIN {X 0,Y 213.977,Z 166.833,A -85,B 0,C 180,E1 -20776.709,E2 -20776.709} C_VEL
LIN {X 0,Y 214.193,Z 166.806,A -85,B 0,C 180,E1 -20780.559,E2 -20780.559} C_VEL
LIN {X 0,Y 214.245,Z 166.799,A -85,B 0,C 180,E1 -20782.461,E2 -20782.461} C_VEL
LIN {X 0,Y 214.443,Z 166.773,A -85,B 0,C 180,E1 -20788.123,E2 -20788.123} C_VEL
LIN {X 0,Y 214.548,Z 166.76,A -85,B 0,C 180,E1 -20790.001,E2 -20790.001} C_VEL
LIN {X 0,Y 214.444,Z 166.773,A -85,B 0,C 180,E1 -20791.879,E2 -20791.879} C_VEL
LIN {X 0,Y 214.163,Z 166.808,A -85,B 0,C 180,E1 -20793.87,E2 -20793.87} C_VEL
LIN {X 0,Y 215.284,Z 169.911,A -85,B 0,C 180,E1 -20794.166,E2 -20794.166} C_VEL
LIN {X 0,Y 222.76,Z 185.459,A -85,B 0,C 180,E1 -20795.768,E2 -20795.768} C_VEL
LIN {X 0,Y 228.82,Z 200.876,A -85,B 0,C 180,E1 -20797.097,E2 -20797.097} C_VEL
LIN {X 0,Y 230.038,Z 204.442,A -85,B 0,C 180,E1 -20797.372,E2 -20797.372} C_VEL
LIN {X 0,Y 227.15,Z 268.994,A -85,B 0,C 180,E1 -20799.578,E2 -20799.578} C_VEL
LIN {X 0,Y 226.057,Z 282.56,A -85,B 0,C 180,E1 -20800.39,E2 -20800.39} C_VEL
LIN {X 0,Y 224.871,Z 294.963,A -85,B 0,C 180,E1 -20801.494,E2 -20801.494} C_VEL
LIN {X 0,Y 223.257,Z 307.024,A -85,B 0,C 180,E1 -20802.939,E2 -20802.939} C_VEL
LIN {X 0,Y 221.288,Z 318.596,A -85,B 0,C 180,E1 -20804.72,E2 -20804.72} C_VEL
LIN {X 0,Y 219.343,Z 329.022,A -85,B 0,C 180,E1 -20806.762,E2 -20806.762} C_VEL
LIN {X 0,Y 217.386,Z 338.992,A -85,B 0,C 180,E1 -20809.235,E2 -20809.235} C_VEL
LIN {X 0,Y 215.593,Z 347.919,A -85,B 0,C 180,E1 -20812.018,E2 -20812.018} C_VEL
LIN {X 0,Y 214.154,Z 354.987,A -85,B 0,C 180,E1 -20814.82,E2 -20814.82} C_VEL
LIN {X 0,Y 213.082,Z 360.391,A -85,B 0,C 180,E1 -20817.502,E2 -20817.502} C_VEL
LIN {X 0,Y 212.227,Z 365.196,A -85,B 0,C 180,E1 -20820.573,E2 -20820.573} C_VEL
LIN {X 0,Y 211.546,Z 368.927,A -85,B 0,C 180,E1 -20823.847,E2 -20823.847} C_VEL
LIN {X 0,Y 211.283,Z 371.3,A -85,B 0,C 180,E1 -20827.032,E2 -20827.032} C_VEL
LIN {X 0,Y 211.416,Z 372.495,A -85,B 0,C 180,E1 -20830.132,E2 -20830.132} C_VEL
LIN {X 0,Y 211.891,Z 372.637,A -85,B 0,C 180,E1 -20833.141,E2 -20833.141} C_VEL
LIN {X 0,Y 212.865,Z 371.57,A -85,B 0,C 180,E1 -20836.583,E2 -20836.583} C_VEL
LIN {X 0,Y 214.56,Z 368.857,A -85,B 0,C 180,E1 -20840.333,E2 -20840.333} C_VEL
LIN {X 0,Y 216.045,Z 366.058,A -85,B 0,C 180,E1 -20842.844,E2 -20842.844} C_VEL
LIN {X 0,Y 218.432,Z 361.283,A -85,B 0,C 180,E1 -20845.982,E2 -20845.982} C_VEL
LIN {X 0,Y 221.359,Z 355.059,A -85,B 0,C 180,E1 -20849.009,E2 -20849.009} C_VEL
LIN {X 0,Y 224.098,Z 348.702,A -85,B 0,C 180,E1 -20851.418,E2 -20851.418} C_VEL
LIN {X 0,Y 227.658,Z 339.936,A -85,B 0,C 180,E1 -20854.018,E2 -20854.018} C_VEL
LIN {X 0,Y 230.74,Z 331.399,A -85,B 0,C 180,E1 -20856.032,E2 -20856.032} C_VEL
LIN {X 0,Y 234.216,Z 320.572,A -85,B 0,C 180,E1 -20858.044,E2 -20858.044} C_VEL
LIN {X 0,Y 237.131,Z 309.455,A -85,B 0,C 180,E1 -20859.667,E2 -20859.667} C_VEL
LIN {X 0,Y 239.648,Z 298.116,A -85,B 0,C 180,E1 -20860.941,E2 -20860.941} C_VEL
LIN {X 0,Y 241.734,Z 285.581,A -85,B 0,C 180,E1 -20862.004,E2 -20862.004} C_VEL
LIN {X 0,Y 243.281,Z 272.642,A -85,B 0,C 180,E1 -20862.752,E2 -20862.752} C_VEL
LIN {X 0,Y 245.461,Z 242.15,A -85,B 0,C 180,E1 -20863.778,E2 -20863.778} C_VEL
LIN {X 0,Y 246.905,Z 218.32,A -85,B 0,C 180,E1 -20864.575,E2 -20864.575} C_VEL
LIN {X 0,Y 241.347,Z 206.583,A -85,B 0,C 180,E1 -20866.569,E2 -20866.569} C_VEL
LIN {X 0,Y 236.579,Z 198.08,A -85,B 0,C 180,E1 -20868.378,E2 -20868.378} C_VEL
LIN {X 0,Y 231.197,Z 190.092,A -85,B 0,C 180,E1 -20870.542,E2 -20870.542} C_VEL
LIN {X 0,Y 228.503,Z 186.145,A -85,B 0,C 180,E1 -20871.739,E2 -20871.739} C_VEL
LIN {X 0,Y 225.671,Z 182.127,A -85,B 0,C 180,E1 -20873.07,E2 -20873.07} C_VEL
LIN {X 0,Y 223.298,Z 179.092,A -85,B 0,C 180,E1 -20874.243,E2 -20874.243} C_VEL
LIN {X 0,Y 222.512,Z 177.792,A -85,B 0,C 180,E1 -20874.677,E2 -20874.677} C_VEL
LIN {X 0,Y 219.886,Z 175.318,A -85,B 0,C 180,E1 -20876.049,E2 -20876.049} C_VEL
LIN {X 0,Y 218.427,Z 172.417,A -85,B 0,C 180,E1 -20876.977,E2 -20876.977} C_VEL
LIN {X 0,Y 216.166,Z 170.601,A -85,B 0,C 180,E1 -20878.313,E2 -20878.313} C_VEL
LIN {X 0,Y 214.852,Z 168.404,A -85,B 0,C 180,E1 -20879.24,E2 -20879.24} C_VEL
LIN {X 0,Y 214.471,Z 166.76,A -85,B 0,C 180,E1 -20879.649,E2 -20879.649} C_VEL
LIN {X 0,Y 214.407,Z 166.77,A -85,B 0,C 180,E1 -20881.879,E2 -20881.879} C_VEL
LIN {X 0,Y 214.183,Z 166.792,A -85,B 0,C 180,E1 -20887.543,E2 -20887.543} C_VEL
LIN {X 0,Y 213.986,Z 166.814,A -85,B 0,C 180,E1 -20891.366,E2 -20891.366} C_VEL
LIN {X 0,Y 213.868,Z 166.829,A -85,B 0,C 180,E1 -20895.243,E2 -20895.243} C_VEL
LIN {X 0,Y 213.793,Z 166.84,A -85,B 0,C 180,E1 -20899.193,E2 -20899.193} C_VEL
LIN {X 0,Y 213.769,Z 166.844,A -85,B 0,C 180,E1 -20903.237,E2 -20903.237} C_VEL
LIN {X 0,Y 213.79,Z 166.842,A -85,B 0,C 180,E1 -20907.427,E2 -20907.427} C_VEL
LIN {X 0,Y 213.755,Z 166.886,A -85,B 0,C 180,E1 -20912.018,E2 -20912.018} C_VEL
LIN {X 0,Y 215.128,Z 170.861,A -85,B 0,C 180,E1 -20916.43,E2 -20916.43} C_VEL
LIN {X 0,Y 215.432,Z 172.317,A -85,B 0,C 180,E1 -20917.394,E2 -20917.394} C_VEL
LIN {X 0,Y 216.021,Z 175.589,A -85,B 0,C 180,E1 -20918.69,E2 -20918.69} C_VEL
LIN {X 0,Y 216.798,Z 179.608,A -85,B 0,C 180,E1 -20919.834,E2 -20919.834} C_VEL
LIN {X 0,Y 219.326,Z 188.168,A -85,B 0,C 180,E1 -20922.006,E2 -20922.006} C_VEL
LIN {X 0,Y 220.601,Z 190.628,A -85,B 0,C 180,E1 -20922.772,E2 -20922.772} C_VEL
LIN {X 0,Y 222.616,Z 193.633,A -85,B 0,C 180,E1 -20923.837,E2 -20923.837} C_VEL
LIN {X 0,Y 226.462,Z 200.168,A -85,B 0,C 180,E1 -20925.751,E2 -20925.751} C_VEL
LIN {X 0,Y 230.923,Z 208.139,A -85,B 0,C 180,E1 -20927.777,E2 -20927.777} C_VEL
LIN {X 0,Y 235.609,Z 218.159,A -85,B 0,C 180,E1 -20929.779,E2 -20929.779} C_VEL
LIN {X 0,Y 239.416,Z 227.273,A -85,B 0,C 180,E1 -20931.311,E2 -20931.311} C_VEL
LIN {X 0,Y 240.678,Z 240.296,A -85,B 0,C 180,E1 -20932.294,E2 -20932.294} C_VEL
LIN {X 0,Y 240.543,Z 244.985,A -85,B 0,C 180,E1 -20932.494,E2 -20932.494} C_VEL
LIN {X 0,Y 237.516,Z 287.073,A -85,B 0,C 180,E1 -20933.911,E2 -20933.911} C_VEL
LIN {X 0,Y 235.655,Z 300.429,A -85,B 0,C 180,E1 -20934.636,E2 -20934.636} C_VEL
LIN {X 0,Y 233.18,Z 312.717,A -85,B 0,C 180,E1 -20935.588,E2 -20935.588} C_VEL
LIN {X 0,Y 230.109,Z 324.972,A -85,B 0,C 180,E1 -20936.91,E2 -20936.91} C_VEL
LIN {X 0,Y 226.656,Z 336.104,A -85,B 0,C 180,E1 -20938.448,E2 -20938.448} C_VEL
LIN {X 0,Y 223.198,Z 346.215,A -85,B 0,C 180,E1 -20940.268,E2 -20940.268} C_VEL
LIN {X 0,Y 219.708,Z 355.382,A -85,B 0,C 180,E1 -20942.365,E2 -20942.365} C_VEL
LIN {X 0,Y 215.92,Z 364.374,A -85,B 0,C 180,E1 -20944.966,E2 -20944.966} C_VEL
LIN {X 0,Y 213.077,Z 371.094,A -85,B 0,C 180,E1 -20947.451,E2 -20947.451} C_VEL
LIN {X 0,Y 210.095,Z 377.558,A -85,B 0,C 180,E1 -20950.456,E2 -20950.456} C_VEL
LIN {X 0,Y 207.935,Z 382.267,A -85,B 0,C 180,E1 -20953.303,E2 -20953.303} C_VEL
LIN {X 0,Y 206.21,Z 385.896,A -85,B 0,C 180,E1 -20956.197,E2 -20956.197} C_VEL
LIN {X 0,Y 205.474,Z 387.762,A -85,B 0,C 180,E1 -20958.156,E2 -20958.156} C_VEL
LIN {X 0,Y 204.567,Z 390.257,A -85,B 0,C 180,E1 -20962.1,E2 -20962.1} C_VEL
LIN {X 0,Y 204.388,Z 391.168,A -85,B 0,C 180,E1 -20965.711,E2 -20965.711} C_VEL
LIN {X 0,Y 204.525,Z 391.021,A -85,B 0,C 180,E1 -20968.03,E2 -20968.03} C_VEL
LIN {X 0,Y 204.672,Z 390.462,A -85,B 0,C 180,E1 -20969.999,E2 -20969.999} C_VEL
LIN {X 0,Y 204.594,Z 389.482,A -85,B 0,C 180,E1 -20971.967,E2 -20971.967} C_VEL
LIN {X 0,Y 204.504,Z 387.356,A -85,B 0,C 180,E1 -20974.704,E2 -20974.704} C_VEL
LIN {X 0,Y 204.668,Z 383.782,A -85,B 0,C 180,E1 -20977.894,E2 -20977.894} C_VEL
LIN {X 0,Y 205.135,Z 379.278,A -85,B 0,C 180,E1 -20980.86,E2 -20980.86} C_VEL
LIN {X 0,Y 206.021,Z 373.517,A -85,B 0,C 180,E1 -20983.814,E2 -20983.814} C_VEL
LIN {X 0,Y 207.467,Z 366.254,A -85,B 0,C 180,E1 -20986.734,E2 -20986.734} C_VEL
LIN {X 0,Y 208.912,Z 358.826,A -85,B 0,C 180,E1 -20989.146,E2 -20989.146} C_VEL
LIN {X 0,Y 210.826,Z 349.837,A -85,B 0,C 180,E1 -20991.511,E2 -20991.511} C_VEL
LIN {X 0,Y 212.869,Z 339.972,A -85,B 0,C 180,E1 -20993.597,E2 -20993.597} C_VEL
LIN {X 0,Y 214.923,Z 329.149,A -85,B 0,C 180,E1 -20995.415,E2 -20995.415} C_VEL
LIN {X 0,Y 216.837,Z 317.039,A -85,B 0,C 180,E1 -20996.984,E2 -20996.984} C_VEL
LIN {X 0,Y 218.46,Z 305.877,A -85,B 0,C 180,E1 -20998.065,E2 -20998.065} C_VEL
LIN {X 0,Y 219.769,Z 292.709,A -85,B 0,C 180,E1 -20998.99,E2 -20998.99} C_VEL
LIN {X 0,Y 220.757,Z 277.142,A -85,B 0,C 180,E1 -20999.632,E2 -20999.632} C_VEL
LIN {X 0,Y 222.371,Z 235.588,A -85,B 0,C 180,E1 -21001.097,E2 -21001.097} C_VEL
LIN {X 0,Y 218.548,Z 203.534,A -85,B 0,C 180,E1 -21002.848,E2 -21002.848} C_VEL
LIN {X 0,Y 210.216,Z 181.561,A -85,B 0,C 180,E1 -21004.859,E2 -21004.859} C_VEL
LIN {X 0,Y 209.269,Z 178.775,A -85,B 0,C 180,E1 -21005.179,E2 -21005.179} C_VEL
LIN {X 0,Y 207.439,Z 170.756,A -85,B 0,C 180,E1 -21008.808,E2 -21008.808} C_VEL
LIN {X 0,Y 206.703,Z 167.741,A -85,B 0,C 180,E1 -21010.24,E2 -21010.24} C_VEL
LIN {X 0,Y 206.633,Z 167.747,A -85,B 0,C 180,E1 -21015.58,E2 -21015.58} C_VEL
LIN {X 0,Y 206.66,Z 167.745,A -85,B 0,C 180,E1 -21019.747,E2 -21019.747} C_VEL
LIN {X 0,Y 206.699,Z 167.738,A -85,B 0,C 180,E1 -21024.687,E2 -21024.687} C_VEL
LIN {X 0,Y 206.723,Z 167.733,A -85,B 0,C 180,E1 -21029.338,E2 -21029.338} C_VEL
LIN {X 0,Y 206.732,Z 167.733,A -85,B 0,C 180,E1 -21033.771,E2 -21033.771} C_VEL
LIN {X 0,Y 206.754,Z 167.729,A -85,B 0,C 180,E1 -21038.042,E2 -21038.042} C_VEL
LIN {X 0,Y 206.825,Z 167.717,A -85,B 0,C 180,E1 -21042.191,E2 -21042.191} C_VEL
LIN {X 0,Y 206.88,Z 167.713,A -85,B 0,C 180,E1 -21046.242,E2 -21046.242} C_VEL
LIN {X 0,Y 207.104,Z 167.683,A -85,B 0,C 180,E1 -21050.23,E2 -21050.23} C_VEL
LIN {X 0,Y 207.166,Z 167.667,A -85,B 0,C 180,E1 -21052.2,E2 -21052.2} C_VEL
LIN {X 0,Y 207.381,Z 167.65,A -85,B 0,C 180,E1 -21058.057,E2 -21058.057} C_VEL
LIN {X 0,Y 207.517,Z 167.63,A -85,B 0,C 180,E1 -21059.999,E2 -21059.999} C_VEL
LIN {X 0,Y 207.38,Z 167.639,A -85,B 0,C 180,E1 -21061.941,E2 -21061.941} C_VEL
LIN {X 0,Y 207.164,Z 167.678,A -85,B 0,C 180,E1 -21067.798,E2 -21067.798} C_VEL
LIN {X 0,Y 206.978,Z 167.695,A -85,B 0,C 180,E1 -21071.754,E2 -21071.754} C_VEL
LIN {X 0,Y 206.863,Z 167.707,A -85,B 0,C 180,E1 -21075.77,E2 -21075.77} C_VEL
LIN {X 0,Y 206.787,Z 167.725,A -85,B 0,C 180,E1 -21079.868,E2 -21079.868} C_VEL
LIN {X 0,Y 206.763,Z 167.717,A -85,B 0,C 180,E1 -21084.071,E2 -21084.071} C_VEL
LIN {X 0,Y 206.74,Z 167.726,A -85,B 0,C 180,E1 -21088.418,E2 -21088.418} C_VEL
LIN {X 0,Y 206.705,Z 167.73,A -85,B 0,C 180,E1 -21092.955,E2 -21092.955} C_VEL
LIN {X 0,Y 206.741,Z 167.719,A -85,B 0,C 180,E1 -21097.725,E2 -21097.725} C_VEL
LIN {X 0,Y 206.75,Z 167.728,A -85,B 0,C 180,E1 -21101.598,E2 -21101.598} C_VEL
LIN {X 0,Y 206.741,Z 167.722,A -85,B 0,C 180,E1 -21105.55,E2 -21105.55} C_VEL
LIN {X 0,Y 206.749,Z 167.731,A -85,B 0,C 180,E1 -21109.771,E2 -21109.771} C_VEL
LIN {X 0,Y 206.741,Z 167.729,A -85,B 0,C 180,E1 -21112.275,E2 -21112.275} C_VEL
LIN {X 0,Y 206.705,Z 167.734,A -85,B 0,C 180,E1 -21117.045,E2 -21117.045} C_VEL
LIN {X 0,Y 206.762,Z 167.729,A -85,B 0,C 180,E1 -21122.097,E2 -21122.097} C_VEL
LIN {X 0,Y 206.781,Z 167.725,A -85,B 0,C 180,E1 -21126.584,E2 -21126.584} C_VEL
LIN {X 0,Y 206.869,Z 167.716,A -85,B 0,C 180,E1 -21132.197,E2 -21132.197} C_VEL
LIN {X 0,Y 206.91,Z 167.713,A -85,B 0,C 180,E1 -21136.246,E2 -21136.246} C_VEL
LIN {X 0,Y 207.129,Z 167.685,A -85,B 0,C 180,E1 -21140.234,E2 -21140.234} C_VEL
LIN {X 0,Y 207.185,Z 167.678,A -85,B 0,C 180,E1 -21142.203,E2 -21142.203} C_VEL
LIN {X 0,Y 207.38,Z 167.653,A -85,B 0,C 180,E1 -21148.059,E2 -21148.059} C_VEL
LIN {X 0,Y 207.512,Z 167.636,A -85,B 0,C 180,E1 -21150.001,E2 -21150.001} C_VEL
LIN {X 0,Y 207.204,Z 167.673,A -85,B 0,C 180,E1 -21152.917,E2 -21152.917} C_VEL
LIN {X 0,Y 208.321,Z 170.76,A -85,B 0,C 180,E1 -21153.24,E2 -21153.24} C_VEL
LIN {X 0,Y 216.918,Z 188.75,A -85,B 0,C 180,E1 -21155.169,E2 -21155.169} C_VEL
LIN {X 0,Y 222.847,Z 204.005,A -85,B 0,C 180,E1 -21156.521,E2 -21156.521} C_VEL
LIN {X 0,Y 223.535,Z 206.339,A -85,B 0,C 180,E1 -21156.696,E2 -21156.696} C_VEL
LIN {X 0,Y 220.537,Z 269.839,A -85,B 0,C 180,E1 -21158.931,E2 -21158.931} C_VEL
LIN {X 0,Y 219.45,Z 282.882,A -85,B 0,C 180,E1 -21159.739,E2 -21159.739} C_VEL
LIN {X 0,Y 218.145,Z 295.666,A -85,B 0,C 180,E1 -21160.912,E2 -21160.912} C_VEL
LIN {X 0,Y 216.528,Z 307.331,A -85,B 0,C 180,E1 -21162.354,E2 -21162.354} C_VEL
LIN {X 0,Y 214.47,Z 319.138,A -85,B 0,C 180,E1 -21164.228,E2 -21164.228} C_VEL
LIN {X 0,Y 212.428,Z 329.711,A -85,B 0,C 180,E1 -21166.378,E2 -21166.378} C_VEL
LIN {X 0,Y 210.34,Z 339.924,A -85,B 0,C 180,E1 -21169.014,E2 -21169.014} C_VEL
LIN {X 0,Y 208.564,Z 348.369,A -85,B 0,C 180,E1 -21171.758,E2 -21171.758} C_VEL
LIN {X 0,Y 207.134,Z 355.218,A -85,B 0,C 180,E1 -21174.561,E2 -21174.561} C_VEL
LIN {X 0,Y 205.964,Z 360.895,A -85,B 0,C 180,E1 -21177.481,E2 -21177.481} C_VEL
LIN {X 0,Y 205.015,Z 366.034,A -85,B 0,C 180,E1 -21180.946,E2 -21180.946} C_VEL
LIN {X 0,Y 204.362,Z 369.645,A -85,B 0,C 180,E1 -21184.377,E2 -21184.377} C_VEL
LIN {X 0,Y 204.196,Z 371.839,A -85,B 0,C 180,E1 -21187.666,E2 -21187.666} C_VEL
LIN {X 0,Y 204.412,Z 372.891,A -85,B 0,C 180,E1 -21190.854,E2 -21190.854} C_VEL
LIN {X 0,Y 204.979,Z 372.923,A -85,B 0,C 180,E1 -21193.946,E2 -21193.946} C_VEL
LIN {X 0,Y 205.88,Z 372.015,A -85,B 0,C 180,E1 -21196.944,E2 -21196.944} C_VEL
LIN {X 0,Y 207.186,Z 370.188,A -85,B 0,C 180,E1 -21199.873,E2 -21199.873} C_VEL
LIN {X 0,Y 209.437,Z 366.331,A -85,B 0,C 180,E1 -21203.647,E2 -21203.647} C_VEL
LIN {X 0,Y 212.295,Z 360.989,A -85,B 0,C 180,E1 -21207.205,E2 -21207.205} C_VEL
LIN {X 0,Y 215.49,Z 354.592,A -85,B 0,C 180,E1 -21210.279,E2 -21210.279} C_VEL
LIN {X 0,Y 218.671,Z 347.601,A -85,B 0,C 180,E1 -21212.887,E2 -21212.887} C_VEL
LIN {X 0,Y 222.13,Z 339.395,A -85,B 0,C 180,E1 -21215.297,E2 -21215.297} C_VEL
LIN {X 0,Y 225.497,Z 330.428,A -85,B 0,C 180,E1 -21217.389,E2 -21217.389} C_VEL
LIN {X 0,Y 229.061,Z 319.592,A -85,B 0,C 180,E1 -21219.36,E2 -21219.36} C_VEL
LIN {X 0,Y 231.977,Z 309.031,A -85,B 0,C 180,E1 -21220.888,E2 -21220.888} C_VEL
LIN {X 0,Y 234.752,Z 296.728,A -85,B 0,C 180,E1 -21222.257,E2 -21222.257} C_VEL
LIN {X 0,Y 236.772,Z 284.579,A -85,B 0,C 180,E1 -21223.265,E2 -21223.265} C_VEL
LIN {X 0,Y 238.277,Z 272.556,A -85,B 0,C 180,E1 -21223.946,E2 -21223.946} C_VEL
LIN {X 0,Y 241.691,Z 225.695,A -85,B 0,C 180,E1 -21225.508,E2 -21225.508} C_VEL
LIN {X 0,Y 241.862,Z 220.967,A -85,B 0,C 180,E1 -21225.702,E2 -21225.702} C_VEL
LIN {X 0,Y 237.144,Z 210.765,A -85,B 0,C 180,E1 -21227.516,E2 -21227.516} C_VEL
LIN {X 0,Y 232.269,Z 202.05,A -85,B 0,C 180,E1 -21229.481,E2 -21229.481} C_VEL
LIN {X 0,Y 225.975,Z 192.494,A -85,B 0,C 180,E1 -21232.263,E2 -21232.263} C_VEL
LIN {X 0,Y 222.862,Z 188.11,A -85,B 0,C 180,E1 -21233.778,E2 -21233.778} C_VEL
LIN {X 0,Y 220.305,Z 184.477,A -85,B 0,C 180,E1 -21235.154,E2 -21235.154} C_VEL
LIN {X 0,Y 217.169,Z 181.049,A -85,B 0,C 180,E1 -21236.894,E2 -21236.894} C_VEL
LIN {X 0,Y 215.913,Z 178.766,A -85,B 0,C 180,E1 -21237.733,E2 -21237.733} C_VEL
LIN {X 0,Y 213.411,Z 176.153,A -85,B 0,C 180,E1 -21239.352,E2 -21239.352} C_VEL
LIN {X 0,Y 211.994,Z 173.398,A -85,B 0,C 180,E1 -21240.476,E2 -21240.476} C_VEL
LIN {X 0,Y 208.641,Z 171.225,A -85,B 0,C 180,E1 -21243.018,E2 -21243.018} C_VEL
LIN {X 0,Y 207.295,Z 168.945,A -85,B 0,C 180,E1 -21244.376,E2 -21244.376} C_VEL
LIN {X 0,Y 207.034,Z 167.697,A -85,B 0,C 180,E1 -21244.869,E2 -21244.869} C_VEL
LIN {X 0,Y 207.127,Z 167.672,A -85,B 0,C 180,E1 -21247.802,E2 -21247.802} C_VEL
LIN {X 0,Y 206.905,Z 167.697,A -85,B 0,C 180,E1 -21251.761,E2 -21251.761} C_VEL
LIN {X 0,Y 206.803,Z 167.709,A -85,B 0,C 180,E1 -21255.777,E2 -21255.777} C_VEL
LIN {X 0,Y 206.713,Z 167.722,A -85,B 0,C 180,E1 -21259.877,E2 -21259.877} C_VEL
LIN {X 0,Y 206.696,Z 167.725,A -85,B 0,C 180,E1 -21264.082,E2 -21264.082} C_VEL
LIN {X 0,Y 206.737,Z 167.781,A -85,B 0,C 180,E1 -21267.077,E2 -21267.077} C_VEL
LIN {X 0,Y 208.058,Z 171.533,A -85,B 0,C 180,E1 -21272.716,E2 -21272.716} C_VEL
LIN {X 0,Y 208.733,Z 173.263,A -85,B 0,C 180,E1 -21274.625,E2 -21274.625} C_VEL
LIN {X 0,Y 212.49,Z 178.694,A -85,B 0,C 180,E1 -21277.677,E2 -21277.677} C_VEL
LIN {X 0,Y 214.247,Z 180.977,A -85,B 0,C 180,E1 -21278.893,E2 -21278.893} C_VEL
LIN {X 0,Y 217.813,Z 186.19,A -85,B 0,C 180,E1 -21281.158,E2 -21281.158} C_VEL
LIN {X 0,Y 219.711,Z 189.23,A -85,B 0,C 180,E1 -21282.271,E2 -21282.271} C_VEL
LIN {X 0,Y 220.601,Z 190.628,A -85,B 0,C 180,E1 -21282.772,E2 -21282.772} C_VEL
LIN {X 0,Y 221.699,Z 193.42,A -85,B 0,C 180,E1 -21283.445,E2 -21283.445} C_VEL
LIN {X 0,Y 222.649,Z 199.339,A -85,B 0,C 180,E1 -21284.246,E2 -21284.246} C_VEL
LIN {X 0,Y 223.614,Z 205.336,A -85,B 0,C 180,E1 -21285.024,E2 -21285.024} C_VEL
LIN {X 0,Y 224.788,Z 208.247,A -85,B 0,C 180,E1 -21285.657,E2 -21285.657} C_VEL
LIN {X 0,Y 229.205,Z 217.031,A -85,B 0,C 180,E1 -21287.744,E2 -21287.744} C_VEL
LIN {X 0,Y 233.929,Z 228.177,A -85,B 0,C 180,E1 -21289.837,E2 -21289.837} C_VEL
LIN {X 0,Y 234.938,Z 231.177,A -85,B 0,C 180,E1 -21290.296,E2 -21290.296} C_VEL
LIN {X 0,Y 235.866,Z 243.043,A -85,B 0,C 180,E1 -21291.183,E2 -21291.183} C_VEL
LIN {X 0,Y 232.669,Z 286.031,A -85,B 0,C 180,E1 -21292.637,E2 -21292.637} C_VEL
LIN {X 0,Y 230.566,Z 300.262,A -85,B 0,C 180,E1 -21293.394,E2 -21293.394} C_VEL
LIN {X 0,Y 227.938,Z 312.946,A -85,B 0,C 180,E1 -21294.409,E2 -21294.409} C_VEL
LIN {X 0,Y 224.718,Z 325.075,A -85,B 0,C 180,E1 -21295.739,E2 -21295.739} C_VEL
LIN {X 0,Y 221.129,Z 336.082,A -85,B 0,C 180,E1 -21297.295,E2 -21297.295} C_VEL
LIN {X 0,Y 217.883,Z 345.055,A -85,B 0,C 180,E1 -21298.928,E2 -21298.928} C_VEL
LIN {X 0,Y 214.192,Z 354.363,A -85,B 0,C 180,E1 -21301.054,E2 -21301.054} C_VEL
LIN {X 0,Y 210.167,Z 363.47,A -85,B 0,C 180,E1 -21303.698,E2 -21303.698} C_VEL
LIN {X 0,Y 206.797,Z 370.787,A -85,B 0,C 180,E1 -21306.428,E2 -21306.428} C_VEL
LIN {X 0,Y 204.32,Z 375.919,A -85,B 0,C 180,E1 -21308.827,E2 -21308.827} C_VEL
LIN {X 0,Y 201.892,Z 380.879,A -85,B 0,C 180,E1 -21311.741,E2 -21311.741} C_VEL
LIN {X 0,Y 199.824,Z 384.746,A -85,B 0,C 180,E1 -21314.704,E2 -21314.704} C_VEL
LIN {X 0,Y 198.502,Z 387.626,A -85,B 0,C 180,E1 -21317.734,E2 -21317.734} C_VEL
LIN {X 0,Y 197.507,Z 390.035,A -85,B 0,C 180,E1 -21321.816,E2 -21321.816} C_VEL
LIN {X 0,Y 197.333,Z 390.647,A -85,B 0,C 180,E1 -21323.865,E2 -21323.865} C_VEL
LIN {X 0,Y 197.329,Z 390.832,A -85,B 0,C 180,E1 -21325.914,E2 -21325.914} C_VEL
LIN {X 0,Y 197.439,Z 390.626,A -85,B 0,C 180,E1 -21327.959,E2 -21327.959} C_VEL
LIN {X 0,Y 197.605,Z 390.027,A -85,B 0,C 180,E1 -21329.999,E2 -21329.999} C_VEL
LIN {X 0,Y 197.505,Z 388.995,A -85,B 0,C 180,E1 -21332.038,E2 -21332.038} C_VEL
LIN {X 0,Y 197.41,Z 387.071,A -85,B 0,C 180,E1 -21334.552,E2 -21334.552} C_VEL
LIN {X 0,Y 197.63,Z 383.13,A -85,B 0,C 180,E1 -21338.177,E2 -21338.177} C_VEL
LIN {X 0,Y 198.125,Z 378.522,A -85,B 0,C 180,E1 -21341.249,E2 -21341.249} C_VEL
LIN {X 0,Y 199.328,Z 371.488,A -85,B 0,C 180,E1 -21344.809,E2 -21344.809} C_VEL
LIN {X 0,Y 200.912,Z 363.842,A -85,B 0,C 180,E1 -21347.822,E2 -21347.822} C_VEL
LIN {X 0,Y 202.521,Z 355.995,A -85,B 0,C 180,E1 -21350.304,E2 -21350.304} C_VEL
LIN {X 0,Y 204.87,Z 345.345,A -85,B 0,C 180,E1 -21352.967,E2 -21352.967} C_VEL
LIN {X 0,Y 207.032,Z 334.498,A -85,B 0,C 180,E1 -21355.107,E2 -21355.107} C_VEL
LIN {X 0,Y 209.067,Z 324.028,A -85,B 0,C 180,E1 -21356.718,E2 -21356.718} C_VEL
LIN {X 0,Y 211.04,Z 311.505,A -85,B 0,C 180,E1 -21358.193,E2 -21358.193} C_VEL
LIN {X 0,Y 212.615,Z 298.469,A -85,B 0,C 180,E1 -21359.315,E2 -21359.315} C_VEL
LIN {X 0,Y 213.772,Z 285.501,A -85,B 0,C 180,E1 -21360.032,E2 -21360.032} C_VEL
LIN {X 0,Y 215.961,Z 237.198,A -85,B 0,C 180,E1 -21361.782,E2 -21361.782} C_VEL
LIN {X 0,Y 212.246,Z 205.735,A -85,B 0,C 180,E1 -21363.55,E2 -21363.55} C_VEL
LIN {X 0,Y 204.59,Z 185.183,A -85,B 0,C 180,E1 -21365.493,E2 -21365.493} C_VEL
LIN {X 0,Y 201.988,Z 178.575,A -85,B 0,C 180,E1 -21366.192,E2 -21366.192} C_VEL
LIN {X 0,Y 200.035,Z 170.277,A -85,B 0,C 180,E1 -21370.127,E2 -21370.127} C_VEL
LIN {X 0,Y 199.617,Z 168.625,A -85,B 0,C 180,E1 -21371.006,E2 -21371.006} C_VEL
LIN {X 0,Y 199.58,Z 168.628,A -85,B 0,C 180,E1 -21375.227,E2 -21375.227} C_VEL
LIN {X 0,Y 199.579,Z 168.623,A -85,B 0,C 180,E1 -21378.004,E2 -21378.004} C_VEL
LIN {X 0,Y 199.61,Z 168.62,A -85,B 0,C 180,E1 -21380.766,E2 -21380.766} C_VEL
LIN {X 0,Y 199.614,Z 168.619,A -85,B 0,C 180,E1 -21385.712,E2 -21385.712} C_VEL
LIN {X 0,Y 199.701,Z 168.61,A -85,B 0,C 180,E1 -21388.136,E2 -21388.136} C_VEL
LIN {X 0,Y 199.686,Z 168.61,A -85,B 0,C 180,E1 -21392.771,E2 -21392.771} C_VEL
LIN {X 0,Y 199.736,Z 168.599,A -85,B 0,C 180,E1 -21397.228,E2 -21397.228} C_VEL
LIN {X 0,Y 199.749,Z 168.599,A -85,B 0,C 180,E1 -21401.796,E2 -21401.796} C_VEL
LIN {X 0,Y 199.817,Z 168.593,A -85,B 0,C 180,E1 -21405.746,E2 -21405.746} C_VEL
LIN {X 0,Y 200.068,Z 168.559,A -85,B 0,C 180,E1 -21409.883,E2 -21409.883} C_VEL
LIN {X 0,Y 200.033,Z 168.56,A -85,B 0,C 180,E1 -21413.949,E2 -21413.949} C_VEL
LIN {X 0,Y 200.32,Z 168.53,A -85,B 0,C 180,E1 -21417.988,E2 -21417.988} C_VEL
LIN {X 0,Y 200.481,Z 168.506,A -85,B 0,C 180,E1 -21419.999,E2 -21419.999} C_VEL
LIN {X 0,Y 200.028,Z 168.558,A -85,B 0,C 180,E1 -21424.028,E2 -21424.028} C_VEL
LIN {X 0,Y 200.108,Z 168.558,A -85,B 0,C 180,E1 -21428.075,E2 -21428.075} C_VEL
LIN {X 0,Y 199.91,Z 168.573,A -85,B 0,C 180,E1 -21432.176,E2 -21432.176} C_VEL
LIN {X 0,Y 199.801,Z 168.588,A -85,B 0,C 180,E1 -21436.343,E2 -21436.343} C_VEL
LIN {X 0,Y 199.705,Z 168.607,A -85,B 0,C 180,E1 -21440.603,E2 -21440.603} C_VEL
LIN {X 0,Y 199.737,Z 168.594,A -85,B 0,C 180,E1 -21443.819,E2 -21443.819} C_VEL
LIN {X 0,Y 199.708,Z 168.601,A -85,B 0,C 180,E1 -21448.386,E2 -21448.386} C_VEL
LIN {X 0,Y 199.66,Z 168.61,A -85,B 0,C 180,E1 -21452.352,E2 -21452.352} C_VEL
LIN {X 0,Y 199.659,Z 168.599,A -85,B 0,C 180,E1 -21456.754,E2 -21456.754} C_VEL
LIN {X 0,Y 199.719,Z 168.6,A -85,B 0,C 180,E1 -21459.3,E2 -21459.3} C_VEL
LIN {X 0,Y 199.698,Z 168.606,A -85,B 0,C 180,E1 -21462.351,E2 -21462.351} C_VEL
LIN {X 0,Y 199.689,Z 168.601,A -85,B 0,C 180,E1 -21465.261,E2 -21465.261} C_VEL
LIN {X 0,Y 199.697,Z 168.604,A -85,B 0,C 180,E1 -21468.037,E2 -21468.037} C_VEL
LIN {X 0,Y 199.72,Z 168.605,A -85,B 0,C 180,E1 -21470.727,E2 -21470.727} C_VEL
LIN {X 0,Y 199.63,Z 168.611,A -85,B 0,C 180,E1 -21475.718,E2 -21475.718} C_VEL
LIN {X 0,Y 199.699,Z 168.609,A -85,B 0,C 180,E1 -21478.138,E2 -21478.138} C_VEL
LIN {X 0,Y 199.682,Z 168.611,A -85,B 0,C 180,E1 -21482.772,E2 -21482.772} C_VEL
LIN {X 0,Y 199.734,Z 168.605,A -85,B 0,C 180,E1 -21487.23,E2 -21487.23} C_VEL
LIN {X 0,Y 199.792,Z 168.599,A -85,B 0,C 180,E1 -21491.758,E2 -21491.758} C_VEL
LIN {X 0,Y 199.844,Z 168.594,A -85,B 0,C 180,E1 -21495.75,E2 -21495.75} C_VEL
LIN {X 0,Y 200.072,Z 168.565,A -85,B 0,C 180,E1 -21499.885,E2 -21499.885} C_VEL
LIN {X 0,Y 200.129,Z 168.558,A -85,B 0,C 180,E1 -21501.926,E2 -21501.926} C_VEL
LIN {X 0,Y 200.32,Z 168.533,A -85,B 0,C 180,E1 -21507.991,E2 -21507.991} C_VEL
LIN {X 0,Y 200.374,Z 168.526,A -85,B 0,C 180,E1 -21511.006,E2 -21511.006} C_VEL
LIN {X 0,Y 200.323,Z 168.538,A -85,B 0,C 180,E1 -21511.949,E2 -21511.949} C_VEL
LIN {X 0,Y 201.342,Z 171.503,A -85,B 0,C 180,E1 -21512.242,E2 -21512.242} C_VEL
LIN {X 0,Y 211.255,Z 192.446,A -85,B 0,C 180,E1 -21514.588,E2 -21514.588} C_VEL
LIN {X 0,Y 216.891,Z 207.169,A -85,B 0,C 180,E1 -21515.925,E2 -21515.925} C_VEL
LIN {X 0,Y 215.194,Z 245.689,A -85,B 0,C 180,E1 -21517.302,E2 -21517.302} C_VEL
LIN {X 0,Y 213.878,Z 271.126,A -85,B 0,C 180,E1 -21518.276,E2 -21518.276} C_VEL
LIN {X 0,Y 212.747,Z 284.43,A -85,B 0,C 180,E1 -21519.156,E2 -21519.156} C_VEL
LIN {X 0,Y 211.291,Z 297.331,A -85,B 0,C 180,E1 -21520.421,E2 -21520.421} C_VEL
LIN {X 0,Y 209.419,Z 310.243,A -85,B 0,C 180,E1 -21522.133,E2 -21522.133} C_VEL
LIN {X 0,Y 207.389,Z 321.001,A -85,B 0,C 180,E1 -21523.973,E2 -21523.973} C_VEL
LIN {X 0,Y 205.146,Z 332.172,A -85,B 0,C 180,E1 -21526.419,E2 -21526.419} C_VEL
LIN {X 0,Y 203.378,Z 340.327,A -85,B 0,C 180,E1 -21528.643,E2 -21528.643} C_VEL
LIN {X 0,Y 201.541,Z 348.753,A -85,B 0,C 180,E1 -21531.48,E2 -21531.48} C_VEL
LIN {X 0,Y 200.202,Z 355.052,A -85,B 0,C 180,E1 -21534.119,E2 -21534.119} C_VEL
LIN {X 0,Y 198.882,Z 361.171,A -85,B 0,C 180,E1 -21537.349,E2 -21537.349} C_VEL
LIN {X 0,Y 198.003,Z 365.922,A -85,B 0,C 180,E1 -21540.619,E2 -21540.619} C_VEL
LIN {X 0,Y 197.402,Z 369.055,A -85,B 0,C 180,E1 -21543.495,E2 -21543.495} C_VEL
LIN {X 0,Y 197.096,Z 371.862,A -85,B 0,C 180,E1 -21547.315,E2 -21547.315} C_VEL
LIN {X 0,Y 197.188,Z 372.922,A -85,B 0,C 180,E1 -21549.908,E2 -21549.908} C_VEL
LIN {X 0,Y 197.567,Z 373.374,A -85,B 0,C 180,E1 -21552.524,E2 -21552.524} C_VEL
LIN {X 0,Y 198.187,Z 373.116,A -85,B 0,C 180,E1 -21555.174,E2 -21555.174} C_VEL
LIN {X 0,Y 199.126,Z 372.175,A -85,B 0,C 180,E1 -21557.889,E2 -21557.889} C_VEL
LIN {X 0,Y 200.575,Z 370.267,A -85,B 0,C 180,E1 -21560.899,E2 -21560.899} C_VEL
LIN {X 0,Y 203.035,Z 366.347,A -85,B 0,C 180,E1 -21564.749,E2 -21564.749} C_VEL
LIN {X 0,Y 205.304,Z 362.43,A -85,B 0,C 180,E1 -21567.468,E2 -21567.468} C_VEL
LIN {X 0,Y 208.002,Z 357.484,A -85,B 0,C 180,E1 -21570.126,E2 -21570.126} C_VEL
LIN {X 0,Y 211.543,Z 350.377,A -85,B 0,C 180,E1 -21573.101,E2 -21573.101} C_VEL
LIN {X 0,Y 215.577,Z 341.563,A -85,B 0,C 180,E1 -21575.902,E2 -21575.902} C_VEL
LIN {X 0,Y 219.431,Z 332.065,A -85,B 0,C 180,E1 -21578.255,E2 -21578.255} C_VEL
LIN {X 0,Y 223.055,Z 321.913,A -85,B 0,C 180,E1 -21580.221,E2 -21580.221} C_VEL
LIN {X 0,Y 226.336,Z 310.777,A -85,B 0,C 180,E1 -21581.911,E2 -21581.911} C_VEL
LIN {X 0,Y 229.246,Z 298.895,A -85,B 0,C 180,E1 -21583.294,E2 -21583.294} C_VEL
LIN {X 0,Y 231.493,Z 286.718,A -85,B 0,C 180,E1 -21584.363,E2 -21584.363} C_VEL
LIN {X 0,Y 233.203,Z 273.828,A -85,B 0,C 180,E1 -21585.139,E2 -21585.139} C_VEL
LIN {X 0,Y 235.075,Z 250.632,A -85,B 0,C 180,E1 -21585.957,E2 -21585.957} C_VEL
LIN {X 0,Y 236.955,Z 223.616,A -85,B 0,C 180,E1 -21586.871,E2 -21586.871} C_VEL
LIN {X 0,Y 231.946,Z 212.877,A -85,B 0,C 180,E1 -21588.958,E2 -21588.958} C_VEL
LIN {X 0,Y 227.683,Z 205.549,A -85,B 0,C 180,E1 -21590.804,E2 -21590.804} C_VEL
LIN {X 0,Y 222.347,Z 197.401,A -85,B 0,C 180,E1 -21593.337,E2 -21593.337} C_VEL
LIN {X 0,Y 219.989,Z 193.901,A -85,B 0,C 180,E1 -21594.587,E2 -21594.587} C_VEL
LIN {X 0,Y 217.162,Z 190.005,A -85,B 0,C 180,E1 -21596.18,E2 -21596.18} C_VEL
LIN {X 0,Y 214.608,Z 186.869,A -85,B 0,C 180,E1 -21597.719,E2 -21597.719} C_VEL
LIN {X 0,Y 213.389,Z 184.914,A -85,B 0,C 180,E1 -21598.556,E2 -21598.556} C_VEL
LIN {X 0,Y 210.848,Z 181.701,A -85,B 0,C 180,E1 -21600.359,E2 -21600.359} C_VEL
LIN {X 0,Y 209.961,Z 180.057,A -85,B 0,C 180,E1 -21601.103,E2 -21601.103} C_VEL
LIN {X 0,Y 206.817,Z 177.689,A -85,B 0,C 180,E1 -21603.654,E2 -21603.654} C_VEL
LIN {X 0,Y 205.415,Z 175.216,A -85,B 0,C 180,E1 -21605.155,E2 -21605.155} C_VEL
LIN {X 0,Y 205.222,Z 174.635,A -85,B 0,C 180,E1 -21605.406,E2 -21605.406} C_VEL
LIN {X 0,Y 201.689,Z 172.261,A -85,B 0,C 180,E1 -21609.782,E2 -21609.782} C_VEL
LIN {X 0,Y 200.005,Z 169.584,A -85,B 0,C 180,E1 -21613.592,E2 -21613.592} C_VEL
LIN {X 0,Y 199.87,Z 169.165,A -85,B 0,C 180,E1 -21614.25,E2 -21614.25} C_VEL
LIN {X 0,Y 199.862,Z 169.308,A -85,B 0,C 180,E1 -21618.451,E2 -21618.451} C_VEL
LIN {X 0,Y 200.309,Z 170.781,A -85,B 0,C 180,E1 -21624.181,E2 -21624.181} C_VEL
LIN {X 0,Y 200.892,Z 171.831,A -85,B 0,C 180,E1 -21626.212,E2 -21626.212} C_VEL
LIN {X 0,Y 201.794,Z 173.379,A -85,B 0,C 180,E1 -21627.939,E2 -21627.939} C_VEL
LIN {X 0,Y 207.105,Z 180.116,A -85,B 0,C 180,E1 -21634.198,E2 -21634.198} C_VEL
LIN {X 0,Y 210.591,Z 185.265,A -85,B 0,C 180,E1 -21637.162,E2 -21637.162} C_VEL
LIN {X 0,Y 212.058,Z 187.351,A -85,B 0,C 180,E1 -21638.241,E2 -21638.241} C_VEL
LIN {X 0,Y 216.202,Z 193.641,A -85,B 0,C 180,E1 -21640.979,E2 -21640.979} C_VEL
LIN {X 0,Y 219.901,Z 199.712,A -85,B 0,C 180,E1 -21643.139,E2 -21643.139} C_VEL
LIN {X 0,Y 223.214,Z 205.456,A -85,B 0,C 180,E1 -21644.88,E2 -21644.88} C_VEL
LIN {X 0,Y 224.788,Z 208.247,A -85,B 0,C 180,E1 -21645.657,E2 -21645.657} C_VEL
LIN {X 0,Y 226.743,Z 212.339,A -85,B 0,C 180,E1 -21646.623,E2 -21646.623} C_VEL
LIN {X 0,Y 228.514,Z 218.961,A -85,B 0,C 180,E1 -21647.63,E2 -21647.63} C_VEL
LIN {X 0,Y 229.827,Z 228.257,A -85,B 0,C 180,E1 -21648.597,E2 -21648.597} C_VEL
LIN {X 0,Y 230.606,Z 235.923,A -85,B 0,C 180,E1 -21649.277,E2 -21649.277} C_VEL
LIN {X 0,Y 231.105,Z 244.293,A -85,B 0,C 180,E1 -21649.9,E2 -21649.9} C_VEL
LIN {X 0,Y 227.83,Z 285.96,A -85,B 0,C 180,E1 -21651.344,E2 -21651.344} C_VEL
LIN {X 0,Y 225.763,Z 299.366,A -85,B 0,C 180,E1 -21652.06,E2 -21652.06} C_VEL
LIN {X 0,Y 223.298,Z 311.206,A -85,B 0,C 180,E1 -21652.99,E2 -21652.99} C_VEL
LIN {X 0,Y 220.404,Z 322.098,A -85,B 0,C 180,E1 -21654.131,E2 -21654.131} C_VEL
LIN {X 0,Y 216.64,Z 333.57,A -85,B 0,C 180,E1 -21655.689,E2 -21655.689} C_VEL
LIN {X 0,Y 212.763,Z 343.971,A -85,B 0,C 180,E1 -21657.535,E2 -21657.535} C_VEL
LIN {X 0,Y 208.835,Z 353.427,A -85,B 0,C 180,E1 -21659.681,E2 -21659.681} C_VEL
LIN {X 0,Y 204.486,Z 362.62,A -85,B 0,C 180,E1 -21662.354,E2 -21662.354} C_VEL
LIN {X 0,Y 200.823,Z 370.066,A -85,B 0,C 180,E1 -21665.167,E2 -21665.167} C_VEL
LIN {X 0,Y 197.729,Z 376.125,A -85,B 0,C 180,E1 -21668.085,E2 -21668.085} C_VEL
LIN {X 0,Y 195.144,Z 380.972,A -85,B 0,C 180,E1 -21671.086,E2 -21671.086} C_VEL
LIN {X 0,Y 192.967,Z 384.733,A -85,B 0,C 180,E1 -21674.147,E2 -21674.147} C_VEL
LIN {X 0,Y 191.529,Z 387.508,A -85,B 0,C 180,E1 -21677.28,E2 -21677.28} C_VEL
LIN {X 0,Y 190.468,Z 389.81,A -85,B 0,C 180,E1 -21681.511,E2 -21681.511} C_VEL
LIN {X 0,Y 190.239,Z 390.48,A -85,B 0,C 180,E1 -21685.762,E2 -21685.762} C_VEL
LIN {X 0,Y 190.354,Z 390.232,A -85,B 0,C 180,E1 -21687.883,E2 -21687.883} C_VEL
LIN {X 0,Y 190.538,Z 389.59,A -85,B 0,C 180,E1 -21689.999,E2 -21689.999} C_VEL
LIN {X 0,Y 190.42,Z 388.471,A -85,B 0,C 180,E1 -21692.114,E2 -21692.114} C_VEL
LIN {X 0,Y 190.339,Z 386.707,A -85,B 0,C 180,E1 -21694.472,E2 -21694.472} C_VEL
LIN {X 0,Y 190.464,Z 383.713,A -85,B 0,C 180,E1 -21697.419,E2 -21697.419} C_VEL
LIN {X 0,Y 190.911,Z 379.393,A -85,B 0,C 180,E1 -21700.605,E2 -21700.605} C_VEL
LIN {X 0,Y 191.742,Z 373.824,A -85,B 0,C 180,E1 -21703.782,E2 -21703.782} C_VEL
LIN {X 0,Y 193.268,Z 366.859,A -85,B 0,C 180,E1 -21706.911,E2 -21706.911} C_VEL
LIN {X 0,Y 194.968,Z 358.503,A -85,B 0,C 180,E1 -21709.878,E2 -21709.878} C_VEL
LIN {X 0,Y 197.131,Z 349.054,A -85,B 0,C 180,E1 -21712.533,E2 -21712.533} C_VEL
LIN {X 0,Y 199.326,Z 339.165,A -85,B 0,C 180,E1 -21714.751,E2 -21714.751} C_VEL
LIN {X 0,Y 201.48,Z 328.275,A -85,B 0,C 180,E1 -21716.685,E2 -21716.685} C_VEL
LIN {X 0,Y 203.558,Z 316.129,A -85,B 0,C 180,E1 -21718.341,E2 -21718.341} C_VEL
LIN {X 0,Y 205.28,Z 304.909,A -85,B 0,C 180,E1 -21719.48,E2 -21719.48} C_VEL
LIN {X 0,Y 206.607,Z 292.574,A -85,B 0,C 180,E1 -21720.396,E2 -21720.396} C_VEL
LIN {X 0,Y 207.594,Z 278.096,A -85,B 0,C 180,E1 -21721.05,E2 -21721.05} C_VEL
LIN {X 0,Y 209.383,Z 237.113,A -85,B 0,C 180,E1 -21722.576,E2 -21722.576} C_VEL
LIN {X 0,Y 205.882,Z 207.496,A -85,B 0,C 180,E1 -21724.316,E2 -21724.316} C_VEL
LIN {X 0,Y 197.417,Z 185.021,A -85,B 0,C 180,E1 -21726.571,E2 -21726.571} C_VEL
LIN {X 0,Y 194.684,Z 178.162,A -85,B 0,C 180,E1 -21727.366,E2 -21727.366} C_VEL
LIN {X 0,Y 192.55,Z 169.504,A -85,B 0,C 180,E1 -21731.724,E2 -21731.724} C_VEL
LIN {X 0,Y 192.491,Z 169.508,A -85,B 0,C 180,E1 -21736.903,E2 -21736.903} C_VEL
LIN {X 0,Y 192.551,Z 169.499,A -85,B 0,C 180,E1 -21741.647,E2 -21741.647} C_VEL
LIN {X 0,Y 192.599,Z 169.494,A -85,B 0,C 180,E1 -21746.813,E2 -21746.813} C_VEL
LIN {X 0,Y 192.664,Z 169.484,A -85,B 0,C 180,E1 -21751.691,E2 -21751.691} C_VEL
LIN {X 0,Y 192.705,Z 169.472,A -85,B 0,C 180,E1 -21756.347,E2 -21756.347} C_VEL
LIN {X 0,Y 192.698,Z 169.479,A -85,B 0,C 180,E1 -21761.485,E2 -21761.485} C_VEL
LIN {X 0,Y 192.741,Z 169.471,A -85,B 0,C 180,E1 -21765.211,E2 -21765.211} C_VEL
LIN {X 0,Y 192.979,Z 169.443,A -85,B 0,C 180,E1 -21769.507,E2 -21769.507} C_VEL
LIN {X 0,Y 193.06,Z 169.424,A -85,B 0,C 180,E1 -21771.626,E2 -21771.626} C_VEL
LIN {X 0,Y 193.262,Z 169.409,A -85,B 0,C 180,E1 -21777.915,E2 -21777.915} C_VEL
LIN {X 0,Y 193.444,Z 169.383,A -85,B 0,C 180,E1 -21779.999,E2 -21779.999} C_VEL
LIN {X 0,Y 192.975,Z 169.437,A -85,B 0,C 180,E1 -21784.176,E2 -21784.176} C_VEL
LIN {X 0,Y 193.059,Z 169.437,A -85,B 0,C 180,E1 -21788.372,E2 -21788.372} C_VEL
LIN {X 0,Y 192.85,Z 169.447,A -85,B 0,C 180,E1 -21792.629,E2 -21792.629} C_VEL
LIN {X 0,Y 192.751,Z 169.474,A -85,B 0,C 180,E1 -21798.562,E2 -21798.562} C_VEL
LIN {X 0,Y 192.663,Z 169.469,A -85,B 0,C 180,E1 -21804.226,E2 -21804.226} C_VEL
LIN {X 0,Y 192.646,Z 169.482,A -85,B 0,C 180,E1 -21808.892,E2 -21808.892} C_VEL
LIN {X 0,Y 192.596,Z 169.487,A -85,B 0,C 180,E1 -21813.185,E2 -21813.185} C_VEL
LIN {X 0,Y 192.624,Z 169.481,A -85,B 0,C 180,E1 -21818.333,E2 -21818.333} C_VEL
LIN {X 0,Y 192.63,Z 169.485,A -85,B 0,C 180,E1 -21823.141,E2 -21823.141} C_VEL
LIN {X 0,Y 192.63,Z 169.479,A -85,B 0,C 180,E1 -21826.859,E2 -21826.859} C_VEL
LIN {X 0,Y 192.624,Z 169.491,A -85,B 0,C 180,E1 -21831.667,E2 -21831.667} C_VEL
LIN {X 0,Y 192.603,Z 169.491,A -85,B 0,C 180,E1 -21837.06,E2 -21837.06} C_VEL
LIN {X 0,Y 192.66,Z 169.488,A -85,B 0,C 180,E1 -21841.693,E2 -21841.693} C_VEL
LIN {X 0,Y 192.701,Z 169.479,A -85,B 0,C 180,E1 -21846.349,E2 -21846.349} C_VEL
LIN {X 0,Y 192.728,Z 169.481,A -85,B 0,C 180,E1 -21851.458,E2 -21851.458} C_VEL
LIN {X 0,Y 192.768,Z 169.475,A -85,B 0,C 180,E1 -21855.215,E2 -21855.215} C_VEL
LIN {X 0,Y 193.016,Z 169.445,A -85,B 0,C 180,E1 -21859.512,E2 -21859.512} C_VEL
LIN {X 0,Y 193.002,Z 169.446,A -85,B 0,C 180,E1 -21863.73,E2 -21863.73} C_VEL
LIN {X 0,Y 193.262,Z 169.412,A -85,B 0,C 180,E1 -21867.917,E2 -21867.917} C_VEL
LIN {X 0,Y 193.35,Z 169.401,A -85,B 0,C 180,E1 -21870.88,E2 -21870.88} C_VEL
LIN {X 0,Y 194.476,Z 172.459,A -85,B 0,C 180,E1 -21871.214,E2 -21871.214} C_VEL
LIN {X 0,Y 205.308,Z 195.417,A -85,B 0,C 180,E1 -21873.899,E2 -21873.899} C_VEL
LIN {X 0,Y 210.49,Z 208.897,A -85,B 0,C 180,E1 -21875.188,E2 -21875.188} C_VEL
LIN {X 0,Y 207.408,Z 270.467,A -85,B 0,C 180,E1 -21877.494,E2 -21877.494} C_VEL
LIN {X 0,Y 206.248,Z 283.744,A -85,B 0,C 180,E1 -21878.37,E2 -21878.37} C_VEL
LIN {X 0,Y 205.005,Z 295.101,A -85,B 0,C 180,E1 -21879.46,E2 -21879.46} C_VEL
LIN {X 0,Y 203.291,Z 306.917,A -85,B 0,C 180,E1 -21880.962,E2 -21880.962} C_VEL
LIN {X 0,Y 201.226,Z 318.002,A -85,B 0,C 180,E1 -21882.776,E2 -21882.776} C_VEL
LIN {X 0,Y 198.933,Z 329.173,A -85,B 0,C 180,E1 -21885.104,E2 -21885.104} C_VEL
LIN {X 0,Y 196.859,Z 338.8,A -85,B 0,C 180,E1 -21887.667,E2 -21887.667} C_VEL
LIN {X 0,Y 194.791,Z 347.92,A -85,B 0,C 180,E1 -21890.721,E2 -21890.721} C_VEL
LIN {X 0,Y 193.308,Z 354.702,A -85,B 0,C 180,E1 -21893.575,E2 -21893.575} C_VEL
LIN {X 0,Y 192.238,Z 359.444,A -85,B 0,C 180,E1 -21896.023,E2 -21896.023} C_VEL
LIN {X 0,Y 191.465,Z 363.436,A -85,B 0,C 180,E1 -21898.503,E2 -21898.503} C_VEL
LIN {X 0,Y 190.572,Z 367.795,A -85,B 0,C 180,E1 -21901.986,E2 -21901.986} C_VEL
LIN {X 0,Y 190.046,Z 370.949,A -85,B 0,C 180,E1 -21905.556,E2 -21905.556} C_VEL
LIN {X 0,Y 190.047,Z 372.858,A -85,B 0,C 180,E1 -21909.053,E2 -21909.053} C_VEL
LIN {X 0,Y 190.445,Z 373.657,A -85,B 0,C 180,E1 -21912.435,E2 -21912.435} C_VEL
LIN {X 0,Y 191.253,Z 373.463,A -85,B 0,C 180,E1 -21915.719,E2 -21915.719} C_VEL
LIN {X 0,Y 192.911,Z 371.82,A -85,B 0,C 180,E1 -21919.914,E2 -21919.914} C_VEL
LIN {X 0,Y 195.213,Z 368.691,A -85,B 0,C 180,E1 -21923.831,E2 -21923.831} C_VEL
LIN {X 0,Y 197.357,Z 365.37,A -85,B 0,C 180,E1 -21926.674,E2 -21926.674} C_VEL
LIN {X 0,Y 200.673,Z 359.921,A -85,B 0,C 180,E1 -21930.091,E2 -21930.091} C_VEL
LIN {X 0,Y 204.466,Z 352.979,A -85,B 0,C 180,E1 -21933.343,E2 -21933.343} C_VEL
LIN {X 0,Y 208.421,Z 345.089,A -85,B 0,C 180,E1 -21936.133,E2 -21936.133} C_VEL
LIN {X 0,Y 212.537,Z 335.885,A -85,B 0,C 180,E1 -21938.671,E2 -21938.671} C_VEL
LIN {X 0,Y 216.081,Z 326.944,A -85,B 0,C 180,E1 -21940.603,E2 -21940.603} C_VEL
LIN {X 0,Y 219.612,Z 316.528,A -85,B 0,C 180,E1 -21942.387,E2 -21942.387} C_VEL
LIN {X 0,Y 222.879,Z 304.976,A -85,B 0,C 180,E1 -21943.93,E2 -21943.93} C_VEL
LIN {X 0,Y 225.44,Z 293.57,A -85,B 0,C 180,E1 -21945.113,E2 -21945.113} C_VEL
LIN {X 0,Y 227.544,Z 281.093,A -85,B 0,C 180,E1 -21946.052,E2 -21946.052} C_VEL
LIN {X 0,Y 228.989,Z 268.979,A -85,B 0,C 180,E1 -21946.646,E2 -21946.646} C_VEL
LIN {X 0,Y 232.248,Z 226.433,A -85,B 0,C 180,E1 -21948.089,E2 -21948.089} C_VEL
LIN {X 0,Y 227.854,Z 217.003,A -85,B 0,C 180,E1 -21950.029,E2 -21950.029} C_VEL
LIN {X 0,Y 224.038,Z 210.336,A -85,B 0,C 180,E1 -21951.819,E2 -21951.819} C_VEL
LIN {X 0,Y 219.558,Z 203.245,A -85,B 0,C 180,E1 -21954.084,E2 -21954.084} C_VEL
LIN {X 0,Y 217.108,Z 199.569,A -85,B 0,C 180,E1 -21955.456,E2 -21955.456} C_VEL
LIN {X 0,Y 214.727,Z 196.228,A -85,B 0,C 180,E1 -21956.859,E2 -21956.859} C_VEL
LIN {X 0,Y 212.073,Z 192.66,A -85,B 0,C 180,E1 -21958.592,E2 -21958.592} C_VEL
LIN {X 0,Y 210.853,Z 190.881,A -85,B 0,C 180,E1 -21959.465,E2 -21959.465} C_VEL
LIN {X 0,Y 208.393,Z 187.328,A -85,B 0,C 180,E1 -21961.377,E2 -21961.377} C_VEL
LIN {X 0,Y 207.706,Z 186.527,A -85,B 0,C 180,E1 -21961.94,E2 -21961.94} C_VEL
LIN {X 0,Y 204.851,Z 183.928,A -85,B 0,C 180,E1 -21964.476,E2 -21964.476} C_VEL
LIN {X 0,Y 203.381,Z 181.298,A -85,B 0,C 180,E1 -21966.2,E2 -21966.2} C_VEL
LIN {X 0,Y 199.995,Z 178.716,A -85,B 0,C 180,E1 -21970.88,E2 -21970.88} C_VEL
LIN {X 0,Y 198.747,Z 176.174,A -85,B 0,C 180,E1 -21974.333,E2 -21974.333} C_VEL
LIN {X 0,Y 198.018,Z 176.322,A -85,B 0,C 180,E1 -21979.167,E2 -21979.167} C_VEL
LIN {X 0,Y 199.301,Z 178.152,A -85,B 0,C 180,E1 -21985.035,E2 -21985.035} C_VEL
LIN {X 0,Y 200.276,Z 179.821,A -85,B 0,C 180,E1 -21987.143,E2 -21987.143} C_VEL
LIN {X 0,Y 205.308,Z 186.629,A -85,B 0,C 180,E1 -21993.578,E2 -21993.578} C_VEL
LIN {X 0,Y 208.673,Z 191.792,A -85,B 0,C 180,E1 -21996.607,E2 -21996.607} C_VEL
LIN {X 0,Y 210.034,Z 193.962,A -85,B 0,C 180,E1 -21997.67,E2 -21997.67} C_VEL
LIN {X 0,Y 213.806,Z 199.893,A -85,B 0,C 180,E1 -22000.309,E2 -22000.309} C_VEL
LIN {X 0,Y 217.065,Z 205.41,A -85,B 0,C 180,E1 -22002.306,E2 -22002.306} C_VEL
LIN {X 0,Y 220.319,Z 211.338,A -85,B 0,C 180,E1 -22004.144,E2 -22004.144} C_VEL
LIN {X 0,Y 224.753,Z 220.161,A -85,B 0,C 180,E1 -22006.412,E2 -22006.412} C_VEL
LIN {X 0,Y 229.306,Z 230.891,A -85,B 0,C 180,E1 -22008.586,E2 -22008.586} C_VEL
LIN {X 0,Y 230.473,Z 234.312,A -85,B 0,C 180,E1 -22009.145,E2 -22009.145} C_VEL
LIN {X 0,Y 230.606,Z 235.923,A -85,B 0,C 180,E1 -22009.277,E2 -22009.277} C_VEL
LIN {X 0,Y 230.679,Z 239.702,A -85,B 0,C 180,E1 -22009.514,E2 -22009.514} C_VEL
LIN {X 0,Y 229.876,Z 245.536,A -85,B 0,C 180,E1 -22009.601,E2 -22009.601} C_VEL
LIN {X 0,Y 226.251,Z 259.16,A -85,B 0,C 180,E1 -22009.276,E2 -22009.276} C_VEL
LIN {X 0,Y 225.047,Z 265.123,A -85,B 0,C 180,E1 -22009.251,E2 -22009.251} C_VEL
LIN {X 0,Y 224.824,Z 267.129,A -85,B 0,C 180,E1 -22009.298,E2 -22009.298} C_VEL
LIN {X 0,Y 223.05,Z 286.963,A -85,B 0,C 180,E1 -22010.027,E2 -22010.027} C_VEL
LIN {X 0,Y 220.834,Z 300.293,A -85,B 0,C 180,E1 -22010.763,E2 -22010.763} C_VEL
LIN {X 0,Y 218.271,Z 311.714,A -85,B 0,C 180,E1 -22011.696,E2 -22011.696} C_VEL
LIN {X 0,Y 214.762,Z 323.898,A -85,B 0,C 180,E1 -22013.035,E2 -22013.035} C_VEL
LIN {X 0,Y 210.878,Z 334.94,A -85,B 0,C 180,E1 -22014.614,E2 -22014.614} C_VEL
LIN {X 0,Y 206.855,Z 345.008,A -85,B 0,C 180,E1 -22016.487,E2 -22016.487} C_VEL
LIN {X 0,Y 202.781,Z 354.176,A -85,B 0,C 180,E1 -22018.675,E2 -22018.675} C_VEL
LIN {X 0,Y 198.253,Z 363.173,A -85,B 0,C 180,E1 -22021.407,E2 -22021.407} C_VEL
LIN {X 0,Y 194.408,Z 370.469,A -85,B 0,C 180,E1 -22024.289,E2 -22024.289} C_VEL
LIN {X 0,Y 191.172,Z 376.368,A -85,B 0,C 180,E1 -22027.292,E2 -22027.292} C_VEL
LIN {X 0,Y 188.411,Z 381.074,A -85,B 0,C 180,E1 -22030.383,E2 -22030.383} C_VEL
LIN {X 0,Y 186.133,Z 384.722,A -85,B 0,C 180,E1 -22033.548,E2 -22033.548} C_VEL
LIN {X 0,Y 184.578,Z 387.396,A -85,B 0,C 180,E1 -22036.793,E2 -22036.793} C_VEL
LIN {X 0,Y 183.889,Z 388.692,A -85,B 0,C 180,E1 -22038.982,E2 -22038.982} C_VEL
LIN {X 0,Y 183.2,Z 390.033,A -85,B 0,C 180,E1 -22043.39,E2 -22043.39} C_VEL
LIN {X 0,Y 183.154,Z 390.111,A -85,B 0,C 180,E1 -22046.107,E2 -22046.107} C_VEL
LIN {X 0,Y 183.472,Z 389.126,A -85,B 0,C 180,E1 -22049.999,E2 -22049.999} C_VEL
LIN {X 0,Y 183.336,Z 387.944,A -85,B 0,C 180,E1 -22052.196,E2 -22052.196} C_VEL
LIN {X 0,Y 183.254,Z 385.355,A -85,B 0,C 180,E1 -22055.501,E2 -22055.501} C_VEL
LIN {X 0,Y 183.535,Z 381.698,A -85,B 0,C 180,E1 -22058.809,E2 -22058.809} C_VEL
LIN {X 0,Y 184.142,Z 376.86,A -85,B 0,C 180,E1 -22062.116,E2 -22062.116} C_VEL
LIN {X 0,Y 185.298,Z 370.712,A -85,B 0,C 180,E1 -22065.395,E2 -22065.395} C_VEL
LIN {X 0,Y 187.004,Z 363.036,A -85,B 0,C 180,E1 -22068.628,E2 -22068.628} C_VEL
LIN {X 0,Y 188.702,Z 355.285,A -85,B 0,C 180,E1 -22071.245,E2 -22071.245} C_VEL
LIN {X 0,Y 190.979,Z 345.51,A -85,B 0,C 180,E1 -22073.877,E2 -22073.877} C_VEL
LIN {X 0,Y 193.367,Z 334.85,A -85,B 0,C 180,E1 -22076.146,E2 -22076.146} C_VEL
LIN {X 0,Y 195.777,Z 322.957,A -85,B 0,C 180,E1 -22078.108,E2 -22078.108} C_VEL
LIN {X 0,Y 197.883,Z 310.32,A -85,B 0,C 180,E1 -22079.669,E2 -22079.669} C_VEL
LIN {X 0,Y 199.569,Z 297.045,A -85,B 0,C 180,E1 -22080.851,E2 -22080.851} C_VEL
LIN {X 0,Y 200.765,Z 283.803,A -85,B 0,C 180,E1 -22081.599,E2 -22081.599} C_VEL
LIN {X 0,Y 202.927,Z 237.837,A -85,B 0,C 180,E1 -22083.372,E2 -22083.372} C_VEL
LIN {X 0,Y 199.676,Z 209.684,A -85,B 0,C 180,E1 -22085.094,E2 -22085.094} C_VEL
LIN {X 0,Y 191.604,Z 188.224,A -85,B 0,C 180,E1 -22087.329,E2 -22087.329} C_VEL
LIN {X 0,Y 187.296,Z 177.774,A -85,B 0,C 180,E1 -22088.624,E2 -22088.624} C_VEL
LIN {X 0,Y 185.477,Z 170.387,A -85,B 0,C 180,E1 -22092.589,E2 -22092.589} C_VEL
LIN {X 0,Y 185.458,Z 170.384,A -85,B 0,C 180,E1 -22096.989,E2 -22096.989} C_VEL
LIN {X 0,Y 185.468,Z 170.384,A -85,B 0,C 180,E1 -22099.894,E2 -22099.894} C_VEL
LIN {X 0,Y 185.506,Z 170.379,A -85,B 0,C 180,E1 -22102.71,E2 -22102.71} C_VEL
LIN {X 0,Y 185.546,Z 170.374,A -85,B 0,C 180,E1 -22107.974,E2 -22107.974} C_VEL
LIN {X 0,Y 185.581,Z 170.361,A -85,B 0,C 180,E1 -22110.574,E2 -22110.574} C_VEL
LIN {X 0,Y 185.587,Z 170.361,A -85,B 0,C 180,E1 -22115.381,E2 -22115.381} C_VEL
LIN {X 0,Y 185.589,Z 170.367,A -85,B 0,C 180,E1 -22120.072,E2 -22120.072} C_VEL
LIN {X 0,Y 185.67,Z 170.349,A -85,B 0,C 180,E1 -22124.634,E2 -22124.634} C_VEL
LIN {X 0,Y 185.922,Z 170.323,A -85,B 0,C 180,E1 -22129.358,E2 -22129.358} C_VEL
LIN {X 0,Y 185.959,Z 170.311,A -85,B 0,C 180,E1 -22133.489,E2 -22133.489} C_VEL
LIN {X 0,Y 186.206,Z 170.288,A -85,B 0,C 180,E1 -22137.836,E2 -22137.836} C_VEL
LIN {X 0,Y 186.407,Z 170.259,A -85,B 0,C 180,E1 -22139.999,E2 -22139.999} C_VEL
LIN {X 0,Y 185.922,Z 170.315,A -85,B 0,C 180,E1 -22144.335,E2 -22144.335} C_VEL
LIN {X 0,Y 186.006,Z 170.316,A -85,B 0,C 180,E1 -22148.691,E2 -22148.691} C_VEL
LIN {X 0,Y 185.761,Z 170.327,A -85,B 0,C 180,E1 -22153.119,E2 -22153.119} C_VEL
LIN {X 0,Y 185.696,Z 170.349,A -85,B 0,C 180,E1 -22157.623,E2 -22157.623} C_VEL
LIN {X 0,Y 185.6,Z 170.36,A -85,B 0,C 180,E1 -22162.25,E2 -22162.25} C_VEL
LIN {X 0,Y 185.559,Z 170.357,A -85,B 0,C 180,E1 -22167.031,E2 -22167.031} C_VEL
LIN {X 0,Y 185.575,Z 170.362,A -85,B 0,C 180,E1 -22169.492,E2 -22169.492} C_VEL
LIN {X 0,Y 185.518,Z 170.362,A -85,B 0,C 180,E1 -22174.627,E2 -22174.627} C_VEL
LIN {X 0,Y 185.563,Z 170.354,A -85,B 0,C 180,E1 -22177.313,E2 -22177.313} C_VEL
LIN {X 0,Y 185.591,Z 170.363,A -85,B 0,C 180,E1 -22180.77,E2 -22180.77} C_VEL
LIN {X 0,Y 185.583,Z 170.354,A -85,B 0,C 180,E1 -22186.014,E2 -22186.014} C_VEL
LIN {X 0,Y 185.579,Z 170.368,A -85,B 0,C 180,E1 -22189.926,E2 -22189.926} C_VEL
LIN {X 0,Y 185.57,Z 170.365,A -85,B 0,C 180,E1 -22192.704,E2 -22192.704} C_VEL
LIN {X 0,Y 185.541,Z 170.374,A -85,B 0,C 180,E1 -22197.976,E2 -22197.976} C_VEL
LIN {X 0,Y 185.577,Z 170.366,A -85,B 0,C 180,E1 -22200.576,E2 -22200.576} C_VEL
LIN {X 0,Y 185.583,Z 170.37,A -85,B 0,C 180,E1 -22205.383,E2 -22205.383} C_VEL
LIN {X 0,Y 185.671,Z 170.359,A -85,B 0,C 180,E1 -22211.134,E2 -22211.134} C_VEL
LIN {X 0,Y 185.72,Z 170.353,A -85,B 0,C 180,E1 -22214.641,E2 -22214.641} C_VEL
LIN {X 0,Y 185.939,Z 170.328,A -85,B 0,C 180,E1 -22219.329,E2 -22219.329} C_VEL
LIN {X 0,Y 185.966,Z 170.324,A -85,B 0,C 180,E1 -22223.491,E2 -22223.491} C_VEL
LIN {X 0,Y 186.324,Z 170.276,A -85,B 0,C 180,E1 -22229.461,E2 -22229.461} C_VEL
LIN {X 0,Y 186.354,Z 170.273,A -85,B 0,C 180,E1 -22229.731,E2 -22229.731} C_VEL
LIN {X 0,Y 187.473,Z 173.227,A -85,B 0,C 180,E1 -22230.08,E2 -22230.08} C_VEL
LIN {X 0,Y 199.259,Z 198.13,A -85,B 0,C 180,E1 -22233.151,E2 -22233.151} C_VEL
LIN {X 0,Y 203.936,Z 210.179,A -85,B 0,C 180,E1 -22234.363,E2 -22234.363} C_VEL
LIN {X 0,Y 200.943,Z 270.269,A -85,B 0,C 180,E1 -22236.686,E2 -22236.686} C_VEL
LIN {X 0,Y 199.721,Z 283.704,A -85,B 0,C 180,E1 -22237.584,E2 -22237.584} C_VEL
LIN {X 0,Y 198.297,Z 296.118,A -85,B 0,C 180,E1 -22238.812,E2 -22238.812} C_VEL
LIN {X 0,Y 196.586,Z 307.345,A -85,B 0,C 180,E1 -22240.298,E2 -22240.298} C_VEL
LIN {X 0,Y 194.266,Z 319.485,A -85,B 0,C 180,E1 -22242.376,E2 -22242.376} C_VEL
LIN {X 0,Y 192.093,Z 329.558,A -85,B 0,C 180,E1 -22244.569,E2 -22244.569} C_VEL
LIN {X 0,Y 189.945,Z 339.175,A -85,B 0,C 180,E1 -22247.219,E2 -22247.219} C_VEL
LIN {X 0,Y 187.943,Z 347.586,A -85,B 0,C 180,E1 -22250.112,E2 -22250.112} C_VEL
LIN {X 0,Y 186.249,Z 355.067,A -85,B 0,C 180,E1 -22253.343,E2 -22253.343} C_VEL
LIN {X 0,Y 184.925,Z 360.889,A -85,B 0,C 180,E1 -22256.524,E2 -22256.524} C_VEL
LIN {X 0,Y 183.98,Z 365.546,A -85,B 0,C 180,E1 -22259.777,E2 -22259.777} C_VEL
